(* IEC 61131-3 sources: volt/packages/volt-lsp-iec/test-corpus/lenze-mid/Device/Plc Logic/Application/Library Manager/L_MC4P_RoboticHandling (part 2) *)

(* ---- AXES_GROUP_KIN.pou ---- *)
FUNCTION_BLOCK AXES_GROUP_KIN EXTENDS AXES_GROUP_REF
VAR_INPUT
	AGBC_INT : L_MC4P_AxesGroupBasicControl_internal;
	PICKANDPLACEMEMORY : L_MC4P_PickAndPlaceMemory;
	XENABLEPRECONTROL : BOOL := FALSE;
	FBKINCOORDPROVIDERTMPUSE : L_MC4P_KinCoordProvider;
	FBPG : L_MC1P_PosProfiler;
	FBFBPOOLCOLLECTION : L_UBUP_FBPoolCollection;
	ITFFBPOOL : L_UBUP_IFBPool := fbFBPoolCollection;
	ITFJOBRECEIVER : L_UBUP_IJobReceiver;
END_VAR
VAR_OUTPUT
	PAXIS_X : POINTER TO AXIS_REF_VMA;
	PAXIS_Y : POINTER TO AXIS_REF_VMA;
	PAXIS_Z : POINTER TO AXIS_REF_VMA;
	PAXIS_A : POINTER TO AXIS_REF_VMA;
	PAXIS_B : POINTER TO AXIS_REF_VMA;
	PAXIS_C : POINTER TO AXIS_REF_VMA;
	XPATHDYNAMICSAVAILABLE : BOOL;
	LRPATHVELOCITY : LREAL;
	LRPATHACCELERATION : LREAL;
	LRPATHROTVELOCITY : LREAL;
	LRPATHROTACCELERATION : LREAL;
	LRTCPVELOCITY : LREAL;
	LRTCPACCELERATION : LREAL;
	XAXESGROUPISHOMED : BOOL := FALSE;
	XINPOSITION : BOOL := FALSE;
END_VAR
VAR
	SCFBSTORE : L_MC4P_MovePathStore;
	FBMOVEFBPOOL : L_MC4P_MoveFBPool;
	FBAGBCFBPOOL : L_MC4P_AGBCFBPool;
	WCS2MCS : REFERENCE TO L_UMTP_RobotPos;
	MCS2WCS : REFERENCE TO L_UMTP_RobotPos;
	LRACTTIMEOR : REFERENCE TO LREAL;
	LRSETTIMEOR : REFERENCE TO LREAL;
	LRACTTIMEDOR : REFERENCE TO LREAL;
	FBCOORD : L_MC4P_KinCoordProvider;
	FBCOORDACT : L_MC4P_KinCoordProvider;
	XMCSDISPLACEMENTSUPPORTED : BOOL := TRUE;
	XDUALUSELICENSEREQUIRED : BOOL := FALSE;
	XDUALUSELICENSEAVAILABLE : BOOL := FALSE;
	XUSEJACOBI : BOOL := TRUE;
	LWSOURCEOFMOTION : LWORD := 0;
	LWFTRIGSOURCEOFMOTION : LWORD := 0;
	XWCSFILTERAVAILABLE : BOOL;
	XUNSTEADYWCSPOS : BOOL;
	ALRUNSTEADYPOSWCS : ARRAY [1..3] OF LREAL;
	FBORFILTERLEGACY : L_MC4P_FilterORLegacy;
	FBORFILTERFAST : L_MC4P_FilterORFast;
	FBORFILTERCOMBINED : L_MC4P_FilterORCombine;
	FBVT : L_MC4P_VirtualTime;
	LRACTTIMEOR_LASTCYCLE : LREAL;
	LROVRREQUESTED : LREAL := 1.0;
	LROVFADINGTIME : LREAL := 0.5;
	_DWOBJID : DWORD;
	PSCTRAFOINFO_SP : POINTER TO L_MC4P_TrafoInfo;
	SCTRAFOINFO_SP : L_MC4P_TrafoInfo;
	PSCTRAFOINFO_ACT : POINTER TO L_MC4P_TrafoInfo;
	SCTRAFOINFO_ACT : L_MC4P_TrafoInfo;
	XPRECONTROLENABLED : BOOL := FALSE;
	AXMCSAXISACTIVE : ARRAY [1..6] OF BOOL;
	AXACSAXISACTIVE : ARRAY [1..6] OF BOOL;
	AXACSAXISALREADYINUSE : ARRAY [1..12] OF BOOL;
	KINPARAMS : L_MC4P_KinematikParam;
	XKINPARAMSVALID : BOOL := FALSE;
	XKINPARAMSVALIDOLD : BOOL := FALSE;
	XKINPARAMSCHANGED : BOOL := FALSE;
	XKINCONFIGAVAILABLE : BOOL := TRUE;
	WINITCOUNTER : WORD;
	ITFKINPARAMS : L_MC4P_IKinematicParameter;
	ITFTRAFO : L_MC4P_ITrafoInterface;
	ITFFFWDTORQUE : L_MC4P_itfTorquePreControl;
	ITFEXTTORQUE : L_MC4P_itfExtDynamics;
	ITFVISU : L_MC4P_VisuInterface;
	ALRTORQUETMP : ARRAY [1..6] OF LREAL;
	AMC_STOP : ARRAY [13..18] OF L_MC1P.L_MC1P_Stop_Internal;
	AMC_HALT : ARRAY [13..18] OF L_MC1P.L_MC1P_Halt_Internal;
	FBDUMMY : L_MC1P.L_MC1P_Template;
	ASCPCSTRACKINGPARAM : ARRAY [1..16] OF L_MC4P_PCSTrackParam;
	DATAVALIDTRACKINGOLD : BOOL := FALSE;
	ECOORDSYSTEMLASTTARGET : L_MC4P_CoordSystem := L_MC4P_CoordSystem.MCS;
	XREAKTONMCFBERROR : BOOL;
	APCS : ARRAY [1..16] OF L_MC4P_CoordTrafo;
	ATOOL : ARRAY [0..4] OF L_MC4P_ToolTrafo;
	AITOOLBUFFERED : ARRAY [0..4] OF INT;
	WACTIVETOOL : L_MC4P_ToolSystem;
	WBUSYTOOL : L_MC4P_ToolSystem;
	MCS : L_MC4P_CoordTrafo;
	AEJCSTRAVERSINGRANGE : ARRAY [1..6] OF L_MC1P_TraversingRange := [6(L_MC1P_TraversingRange.Limited)];
	ALRAPPLVELLIMITS : ARRAY [1..18] OF LREAL := [18(0)];
	ALRAPPLACCLIMITS : ARRAY [1..18] OF LREAL := [18(0)];
	ALRAPPLJERKLIMITS : ARRAY [1..18] OF LREAL := [18(0)];
	WLOOKAHEADHORIZON : WORD;
	XENABLEFULLBLENDING : BOOL := TRUE;
	XLIMITTANGENTIALROTATION : BOOL;
	LRMAXVELTRANSLATION : LREAL;
	LRMAXACCTRANSLATION : LREAL;
	LRMAXJERKTRANSLATION : LREAL;
	LRMAXVELROTATION : LREAL;
	LRMAXACCROTATION : LREAL;
	LRMAXJERKROTATION : LREAL;
	LRTIMEINLISTMIN : LREAL := 0.5;
	LRLA_SECURECYCLECOUNT : LREAL := 20;
	XSETVALUESAVAILABLE : BOOL := FALSE;
	XUSEREALDRIVESASVIRTUAL : BOOL := FALSE;
	XUSEREALDRIVESASVIRTUALOLD : BOOL := FALSE;
	XWAITFORREALDRIVESDISABLED : BOOL;
	PREPAREPATH : L_MC4P_PreparePath;
	INTERPOLATEPATH : L_MC4P_InterpolatePath;
	XLIMITPATHTOMAINAXES : BOOL := TRUE;
	XINTERRUPTATNEXTBUFFEREDPOS : BOOL := FALSE;
	XERRORSTOPDONE : BOOL;
	AEAXISTYPE : ARRAY [1..24] OF L_MC4P_AxisType := [24(L_MC4P_AxisType.unconnected)];
	ALRSCALEGENERALIZEDFORCETOTORQUE : ARRAY [1..6] OF LREAL := [6(1)];
	ALRSCALETORQUETOGENERALIZEDFORCE : ARRAY [1..6] OF LREAL := [6(1)];
	USINBROFACSAXES : USINT;
	EROTATIONCONVENTION : L_UMTP_RotationConvention := L_UMTP_RotationConvention.XYZ_rotated;
	AXROTANGLESFIXED : ARRAY [1..3] OF BOOL := [FALSE, FALSE, FALSE];
	WGROUPSTATUS : DWORD := 0;
	XSETINPOSITION : BOOL;
	PCONNECTOR_AXIS_X : POINTER TO IoConfigConnector;
	PCONNECTOR_AXIS_Y : POINTER TO IoConfigConnector;
	PCONNECTOR_AXIS_Z : POINTER TO IoConfigConnector;
	PCONNECTOR_AXIS_A : POINTER TO IoConfigConnector;
	PCONNECTOR_AXIS_B : POINTER TO IoConfigConnector;
	PCONNECTOR_AXIS_C : POINTER TO IoConfigConnector;
	APLINKEDAXIS : ARRAY [1..12] OF POINTER TO AXIS_REF;
	ASLINKEDAXISNAME : ARRAY [1..12] OF STRING;
	XACSAXESCONNECTED : BOOL := FALSE;
	XACSAXESCONNECTEDOLD : BOOL := FALSE;
	XGENERICGROUP : BOOL := FALSE;
	PLRDUMMY : POINTER TO LREAL;
	DIRCREATEMOVEPATHDATA : File.DirCreate;
	DIRCREATEDIAGNOSISDATA : File.DirCreate;
	SDIRDIAGNOSISDATA : STRING;
	EJERKMODE : WORD;
	XIGNOREJERK_CP : BOOL := FALSE;
	XIGNOREJERK_PTP : BOOL := FALSE;
	XIGNOREJERK_AUX : BOOL := FALSE;
	DWUNDOBLENDINGCOUNTER : DWORD;
	LRPATHVELOLD : LREAL := 0;
	LRPATHROTVELOLD : LREAL := 0;
	ROTQUAT : ARRAY [1..4] OF LREAL;
	ROTQUATOLD : ARRAY [1..4] OF LREAL;
	ROTMAT_A : ARRAY [1..3, 1..3] OF LREAL;
	ROTMAT_B : ARRAY [1..3, 1..3] OF LREAL;
	ROTMAT_C : ARRAY [1..3, 1..3] OF LREAL;
	ROTMAT_A_OLD : ARRAY [1..3, 1..3] OF LREAL;
	ROTMAT_B_OLD : ARRAY [1..3, 1..3] OF LREAL;
	ROTMAT_C_OLD : ARRAY [1..3, 1..3] OF LREAL;
	APUNKT : LREAL;
	BPUNKT : LREAL;
	CPUNKT : LREAL;
	FBMCDIAGNOSTIC : L_MC4P_MoveFBDiagnostic;
	FBPATHLISTDIAGNOSTIC : L_MC4P_PathListDiagnostic;
	FBTRACELIST : L_MC4P_TraceList;
	FBOBSERVELIMITS : L_MC4P_ObserveLimits;
	DWRUNTIMECNTR : DWORD;
	SCSUPERPOSDATA : L_MC4P_SuperposHandler;
	SCTRACKINGHANDSHAKE : L_MC4P_TrackingHandshake;
	XORIENTATIONCHANGED : BOOL;
	ACSACC : POINTER TO LREAL;
	ACSPOS : POINTER TO LREAL;
	ACSVEL : POINTER TO LREAL;
	ACTIVELIMITS_1 : DWORD;
	ACTIVELIMITS_2 : DWORD;
	ACTUALINTERPOLATEDMOVEFBINSTANCE : STRING;
	ACTUALINTERPOLATEDSEGMENTID : DINT;
	ACTUALINTERPOLATEDSEGMENTTARGETACS : ARRAY [1..6] OF LREAL;
	ACTUALINTERPOLATEDSEGMENTTARGETAUX : ARRAY [1..6] OF LREAL;
	ACTUALINTERPOLATEDSEGMENTTARGETMCS : ARRAY [1..6] OF LREAL;
	ACTUALINTERPOLATEDSEGMENTTARGETWCS : ARRAY [1..6] OF LREAL;
	ACTUALINTERPOLATEDSEGMENTTYPE : L_MC4P_SegmentType;
	ACTUALSEGMENTSTARTPOSWCS : ARRAY [1..6] OF LREAL;
	CHECKWORKSPACE : BOOL;
	CHECKWORKSPACESTEPS : UDINT;
	CLASSID : DINT;
	CONFIGURATION : ARRAY [1..6] OF INT;
	COORDSYSTEMLASTTARGET : L_MC4P_CoordSystem;
	DIGITALSWITCHHANDLER : L_MC4P_IDigSwitchHandling;
	DIM : UDINT;
	ENABLEMCDIAGNOSTIC : BOOL;
	ENABLEOBSERVELIMITS : BOOL;
	ENABLETRACELISTVISU : BOOL;
	FCSACC : POINTER TO LREAL;
	FCSFRAME : POINTER TO L_UMTP_RobotFrame;
	FCSPOS : POINTER TO LREAL;
	FCSVEL : POINTER TO LREAL;
	HOLDOBSERVEDLIMITS : BOOL;
	IGNOREOVERRIDEWAITTIME : BOOL;
	INTERRUPTATNEXTBUFFEREDPOS : BOOL;
	INTERRUPTEDATNEXTBUFFEREDPOS : BOOL;
	JCSACC : POINTER TO LREAL;
	JCSPOS : POINTER TO LREAL;
	JCSVEL : POINTER TO LREAL;
	LA_SECURECYCLECOUNT : LREAL;
	LOWERSYSTEM : UDINT;
	MAXTANGENTROTACC : LREAL;
	MAXTANGENTROTVEL : LREAL;
	MCSACC : POINTER TO LREAL;
	MCSFRAME : POINTER TO L_UMTP_RobotFrame;
	MCSPOS : POINTER TO LREAL;
	MCSVEL : POINTER TO LREAL;
	OBJECTID : DWORD;
	ORIENTATIONCHANGED : BOOL;
	OVRTYPE : L_MC4P_OVRType;
	PATHACCREDUCTIONFACTOR : LREAL;
	PATHLENGTH : LREAL;
	PATHLISTDIAGBUSY : BOOL;
	PATHLISTDIAGDONE : BOOL;
	PATHLISTDIAGENABLE : BOOL;
	PATHLISTDIAGERRORDETECTED : BOOL;
	PATHLISTDIAGNUMOFLISTELEMENTS : INT;
	PATHLISTDIAGREADERRORFILEEXECUTE : BOOL;
	PATHLISTDIAGWRITEFILEBUSY : BOOL;
	PATHLISTDIAGWRITEFILEDONE : BOOL;
	PATHLISTDIAGWRITEFILEERROR : BOOL;
	PATHLISTDIAGWRITEFILEEXECUTE : BOOL;
	REMAININGPATHLENGTH : LREAL;
	REMAININGSEGMENTLENGTH : LREAL;
	RESETOBSERVEDLIMITS : BOOL;
	SEGMENTLENGTH : LREAL;
	STARTWRITINGDIAGNOSTICFILE : BOOL;
	TANGENTIALTRACKINGENABLEPATHREDUCTION : BOOL;
	TIMEINPATHLISTMIN : LREAL;
	TIMEMEASUREMENT : BOOL;
	UPPERSYSTEM : UDINT;
	USEJACOBI : BOOL;
	WCSACC : POINTER TO LREAL;
	WCSFRAME : POINTER TO L_UMTP_RobotFrame;
	WCSPOS : POINTER TO LREAL;
	WCSVEL : POINTER TO LREAL;
	WRITEDIAGNOSTICFILEDONE : BOOL;
END_VAR
END_FUNCTION_BLOCK

METHOD GENERATEHOMINGSTATEAXIS
VAR_INPUT
	XAXESGROUPISHOMEDOLD : BOOL;
END_VAR
END_METHOD

METHOD GETTRACKINGPCS : POINTER TO L_MC4P_PCSTrackParam
VAR_INPUT
	COORDSYSTEM : L_MC4P_CoordSystem;
END_VAR
END_METHOD

METHOD HASAUXAXIS : BOOL
END_METHOD

METHOD HASONLYCROTATION : BOOL
END_METHOD

METHOD HASROTATIONAXIS : BOOL
END_METHOD

METHOD SETCOMMANDEDPOSITION
VAR_IN_OUT
	ALRCOMMANDEDPOSWCS : ARRAY [1..6] OF LREAL;
	ALRCOMMANDEDPOSACS : ARRAY [1..6] OF LREAL;
	ALRCOMMANDEDPOSAUX : ARRAY [1..6] OF LREAL;
END_VAR
END_METHOD

METHOD SETEXTTORQUEITF : L_IE1P_Error
VAR_INPUT
	ITFEXTTORQUE : L_MC4P_itfExtDynamics;
END_VAR
END_METHOD

METHOD SETINPOSPREPARE
END_METHOD

METHOD SETINPOSITION
VAR_INPUT
	XDONE : BOOL;
END_VAR
END_METHOD

METHOD SETKINREF
VAR_INPUT
	KINTRANSFORM : MC_KIN_REF;
END_VAR
END_METHOD

METHOD SETKINTRANSFORM
VAR_INPUT
	TRAFO : L_MC4P_ITrafoInterface;
END_VAR
END_METHOD

METHOD SETPATHINFO
END_METHOD

METHOD SETSTATUSWORD
END_METHOD

METHOD SETTORQUECTRLFB
VAR_INPUT
	FB : L_MC4P_itfTorquePreControl;
END_VAR
END_METHOD

METHOD SETVISUFB
VAR_INPUT
	VISU : L_MC4P_VisuInterface;
END_VAR
END_METHOD

METHOD UPDATESCALEGENERALIZEDFORCETOTORQUE
END_METHOD

METHOD CHECKAXESTRAVERSINGRANGE : L_IE1P_Error
END_METHOD

METHOD CHECKDUALUSE : BOOL
END_METHOD

METHOD CONFIGUREAXESGROUP
END_METHOD

METHOD GETCONFIGURATIONMAINAXIS
VAR_INPUT
	PFATHER : POINTER TO IoConfigConnector;
	NCOUNT : DINT;
END_VAR
END_METHOD

METHOD ADDACSAXESTOGROUP
VAR_INPUT
	WINDEX : WORD;
END_VAR
END_METHOD

METHOD ADDALLMCSAXISTOGROUP
END_METHOD

METHOD CHECKACSCONFIG : BOOL
END_METHOD

METHOD CONFIGUREAXES : L_IE1P_Error
END_METHOD

METHOD GETAXISMCS : BOOL
VAR_INPUT
	PAXISCONNECTOR : POINTER TO IoConfigConnector;
	XCONNECTED : BOOL;
END_VAR
VAR_OUTPUT
	PAXIS : POINTER TO _AXIS_REF_VMA;
END_VAR
END_METHOD

METHOD REGISTERACSAXISINGROUP
VAR_INPUT
	WINDEX : WORD;
END_VAR
END_METHOD

METHOD SETLINKEDAXIS
VAR_INPUT
	WINDEX : WORD;
END_VAR
END_METHOD

METHOD UPDATEVIRTUALMODEACS
VAR_INPUT
	PAXIS : POINTER TO AXIS_REF;
	XVIRTUALMODE : BOOL;
END_VAR
END_METHOD

METHOD MEMORISEIPOVALUES
VAR_INPUT
	ECOORDSYSTEM : L_MC4P_CoordSystem;
END_VAR
END_METHOD

METHOD BACKWARDTRANSFORMATIONTOAXES : L_IE1P_Error
END_METHOD

METHOD BACKWARDTRANSFORMATIONTOAXES_LEGACY : L_IE1P_Error
VAR_OUTPUT
	SCERROR : L_MC4P_ErrorStruct;
END_VAR
VAR_IN_OUT
	FBCOORD : L_MC4P_KinCoordProvider;
END_VAR
END_METHOD

METHOD BACKWARDTRANSFORMATIONTOAXES_USEJACOBI : L_IE1P_Error
VAR_OUTPUT
	SCERROR : L_MC4P_ErrorStruct;
END_VAR
VAR_IN_OUT
	FBCOORD : L_MC4P_KinCoordProvider;
END_VAR
END_METHOD

METHOD CHECKPLAUSIBILITYOFSETVALUES : L_IE1P.L_IE1P_Error
END_METHOD

METHOD CLEARTRACKINGPCSFLAGS
END_METHOD

METHOD CLEARTRACKINGSUPERPOSDATA
END_METHOD

METHOD FORWARDTRANSFORMATIONTOAXES : L_IE1P_Error
VAR_INPUT
	XUSESETVALUES : BOOL;
END_VAR
END_METHOD

METHOD FORWARDTRANSFORMATIONTOAXES_LEGACY : L_IE1P_Error
VAR_INPUT
	XUSESETVALUES : BOOL;
END_VAR
VAR_OUTPUT
	SCERROR : L_MC4P_ErrorStruct;
END_VAR
VAR_IN_OUT
	FBCOORD : L_MC4P_KinCoordProvider;
END_VAR
END_METHOD

METHOD FORWARDTRANSFORMATIONTOAXES_USEJACOBI : L_IE1P_Error
VAR_INPUT
	XUSESETVALUES : BOOL;
END_VAR
VAR_OUTPUT
	SCERROR : L_MC4P_ErrorStruct;
END_VAR
VAR_IN_OUT
	FBCOORD : L_MC4P_KinCoordProvider;
END_VAR
END_METHOD

METHOD GETCOORDTRAFO : POINTER TO L_MC4P_CoordTrafo
VAR_INPUT
	COORDSYSTEM : L_MC4P_CoordSystem;
END_VAR
END_METHOD

METHOD HANDLEUNSTEADYWCSPOS
END_METHOD

METHOD SETUNSTEADYWCSPOS
VAR_INPUT
	ALRUNSTEADYDISTANCE : ARRAY [1..3] OF LREAL;
END_VAR
END_METHOD

METHOD SUPERPOSETRACKINGVALUES
END_METHOD

METHOD TRACKINGSETSETVALUESAVAILABLE
END_METHOD

METHOD GETMAXACCELERATION : LREAL
VAR_INPUT
	IDX : UINT;
	EMAXVALUESOURCE : L_MC4P_MaxValueSource;
END_VAR
END_METHOD

METHOD GETMAXDECELERATION : LREAL
VAR_INPUT
	IDX : UINT;
	EMAXVALUESOURCE : L_MC4P_MaxValueSource;
END_VAR
END_METHOD

METHOD GETMAXJERK : LREAL
VAR_INPUT
	IDX : UINT;
	EMAXVALUESOURCE : L_MC4P_MaxValueSource;
END_VAR
END_METHOD

METHOD GETMAXVELOCITY : LREAL
VAR_INPUT
	IDX : UINT;
	EMAXVALUESOURCE : L_MC4P_MaxValueSource;
END_VAR
END_METHOD

METHOD EQUALS : BOOL
VAR_INPUT
	ITFPROVIDER : L_MC4P_IKinCoordProvider;
	UDISYSTEM : UDINT;
	XPOS : BOOL;
	XVEL : BOOL;
	XACC : BOOL;
END_VAR
END_METHOD

METHOD REQUESTINTERFACE : BOOL
VAR_INPUT
	ID : DINT;
	PITFUNKNOWN : POINTER TO L_UBUP_IUnknown;
END_VAR
END_METHOD

METHOD SETINSTANCESTRINGMOVEPATHSTORE
VAR_INPUT
	SINSTANCESTR : STRING;
END_VAR
END_METHOD

METHOD APPLYOVERRIDE
VAR_IN_OUT
	LRVEL : LREAL;
	LRACC : LREAL;
END_VAR
END_METHOD

METHOD SETTIMEOVERRIDE
VAR_INPUT
	LROVERRIDE : LREAL;
	LRFADINGTIME : LREAL;
END_VAR
END_METHOD

METHOD CALCSCALEFUNCTIONS
VAR_INPUT
	OFFSET : DWORD;
	INDEX : WORD;
END_VAR
END_METHOD

METHOD CHECKPARAMETER : BOOL
END_METHOD

METHOD ISACTIVEMOTIONCOMMAND : BOOL
VAR_INPUT
	ESRCOFCMD : L_MC4P_SourceOfMotionCommand;
END_VAR
END_METHOD

METHOD RELEASEMOTIONCOMMAND : BOOL
VAR_INPUT
	ESRCOFCMD : L_MC4P_SourceOfMotionCommand;
END_VAR
END_METHOD

METHOD REQUESTMOTIONCOMMAND : L_IE1P_Error
VAR_INPUT
	ESRCOFCMD : L_MC4P_SourceOfMotionCommand;
END_VAR
END_METHOD

METHOD RESETSOURCEOFMOTION
END_METHOD

METHOD SETVALUESCALCULATED
END_METHOD

METHOD UPDATESOURCEOFMOTIONCOMMAND : BOOL
END_METHOD

METHOD CALLSTOPPINTERPOLATOR
VAR_INPUT
	LRINPUTDECELERATION : LREAL;
	LRINPUTJERK : LREAL;
END_VAR
VAR_OUTPUT
	XERROR : BOOL;
	EERRORID : L_IE1P_Error;
	DWINTERNALID : DWORD;
	XDONE : BOOL;
END_VAR
END_METHOD

METHOD ERRORSTOP
END_METHOD

METHOD HALTAUX : BOOL
VAR_OUTPUT
	XERROR : BOOL;
END_VAR
END_METHOD

METHOD LEAVEERRORSTOP
END_METHOD

METHOD LEAVEERRORSTOPPREPARE : BOOL
VAR_INPUT
	XLEAVEERRORSTOP : BOOL;
END_VAR
END_METHOD

METHOD STOPAUX : BOOL
VAR_OUTPUT
	XERROR : BOOL;
END_VAR
END_METHOD

METHOD GETPATHCOORDINATESYSTEM
VAR_OUTPUT
	ALRTANGENT : ARRAY [1..3] OF LREAL;
	ALRNORMAL : ARRAY [1..3] OF LREAL;
	ALRBINORMAL : ARRAY [1..3] OF LREAL;
END_VAR
END_METHOD

METHOD BUFFERTOOL : BOOL
VAR_INPUT
	ETOOLSYSTEM : L_MC4P_ToolSystem;
END_VAR
END_METHOD

METHOD CALCTOOLDISTANCE : BOOL
VAR_INPUT
	ETOOL1 : L_MC4P_ToolSystem;
	ETOOL2 : L_MC4P_ToolSystem;
	SCFCSFRAME : REFERENCE TO L_UMTP_RobotFrame;
	SCDISTWCS : REFERENCE TO L_UMTP_RobotPos;
	SCDISTFCS : REFERENCE TO L_UMTP_RobotPos;
END_VAR
END_METHOD

METHOD CLEARTOOLBUFFER : BOOL
END_METHOD

METHOD GETTOOL : POINTER TO L_MC4P_ToolTrafo
VAR_INPUT
	TOOLSYSTEM : L_MC4P_ToolSystem;
END_VAR
END_METHOD

METHOD SETACTIVETOOL : BOOL
VAR_INPUT
	ETOOLSYSTEM : L_MC4P_ToolSystem;
END_VAR
VAR_OUTPUT
	XTOOLCHANGED : BOOL;
END_VAR
END_METHOD

METHOD TOOLPARAMAPPLICABLE : L_IE1P_Error
VAR_INPUT
	ETOOLSYSTEM : L_MC4P_ToolSystem;
	SCTOOLPARAMETER : L_MC4P_TOOL_REF;
END_VAR
END_METHOD

METHOD TOOLROTATIONISIDENTITY : BOOL
VAR_INPUT
	ETOOLSYSTEM : L_MC4P_ToolSystem;
END_VAR
END_METHOD

METHOD AFTERREADINPUTS : INT
END_METHOD

METHOD AFTERWRITEOUTPUTS
END_METHOD

METHOD BEFOREREADINPUTS : INT
END_METHOD

METHOD BEFOREWRITEOUTPUTS
END_METHOD

METHOD CALL_WCSBWO
END_METHOD

METHOD FB_EXIT : BOOL
VAR_INPUT
	BINCOPYCODE : BOOL;
END_VAR
END_METHOD

METHOD INITFORSIMULATIONMODE : BOOL
VAR_INPUT
	WMODULETYPE : UINT;
	DWINSTANCE : UDINT;
	PCONNECTOR : POINTER TO IoConfigConnector;
END_VAR
END_METHOD

METHOD INITIALIZE : UDINT
VAR_INPUT
	WMODULETYPE : UINT;
	DWINSTANCE : UDINT;
	PCONNECTOR : POINTER TO IoConfigConnector;
END_VAR
END_METHOD

METHOD IODRVREADPARAMETER : UDINT
VAR_INPUT
	PCONNECTOR : POINTER TO IoConfigConnector;
	PPARAMETER : POINTER TO IoConfigParameter;
	PDATA : POINTER TO BYTE;
	DWBITSIZE : DWORD;
	DWBITOFFSET : DWORD;
END_VAR
END_METHOD

METHOD IODRVUPDATECONFIGURATION : UDINT
VAR_INPUT
	PCONNECTORLIST : POINTER TO IoConfigConnector;
	NCOUNT : DINT;
END_VAR
END_METHOD

METHOD IODRVWRITEPARAMETER : UDINT
VAR_INPUT
	PCONNECTOR : POINTER TO IoConfigConnector;
	PPARAMETER : POINTER TO IoConfigParameter;
	PDATA : POINTER TO BYTE;
	DWBITSIZE : DWORD;
	DWBITOFFSET : DWORD;
END_VAR
END_METHOD

METHOD FB_INIT : BOOL
VAR_INPUT
	BINITRETAINS : BOOL;
	BINCOPYCODE : BOOL;
END_VAR
END_METHOD

(* ---- AXES_GROUP_REF.pou ---- *)
FUNCTION_BLOCK AXES_GROUP_REF EXTENDS AXES_GROUP_BASE
VAR_INPUT
	EAXESGROUPSTATE : L_MC4P_AxesGroup_State := L_MC4P_AxesGroup_State.GroupDisabled;
	XGROUPENABLE : BOOL;
	ASCERRORINFO : REFERENCE TO ARRAY [0..7] OF L_IE1P_ErrorInformation;
	ASCWARNINGINFO : REFERENCE TO ARRAY [0..7] OF L_IE1P_ErrorInformation;
	FBFUNIDMANAGER : L_MC4P_FunIDManager;
END_VAR
VAR_OUTPUT
	XERROR : BOOL := FALSE;
	XWARNING : BOOL := FALSE;
	EACTIVEERRORID : L_IE1P_Error;
	XGROUPENABLED : BOOL;
	AXESGROUPNAME : STRING;
END_VAR
VAR
	SCPARAMS : L_MC4P_AxesGroupMember;
	XWRITEGROUPPARAMETERDISABLED : BOOL;
	XISAXES_GROUP_KIN : BOOL := FALSE;
	EKINEMATIC : L_MC4P_KinematicType;
	APAXIS : ARRAY [1..18] OF POINTER TO AXIS_REF;
	ERRORMANAGER : L_IE1P_ErrorManager;
	ERRORRESETOCCUREDTIMEWITHOUTLEM : SYSTIME;
	DWGROUPERRORITFID : DWORD;
	ADWAXISERRORITFID : ARRAY [1..18] OF DWORD;
	PSERRORINST : POINTER TO STRING;
	SERRORINST : STRING;
	XENABLELOGENTRY : BOOL := TRUE;
	EAXESGROUPSTATEOLD : L_MC4P_AxesGroup_State := L_MC4P_AxesGroup_State.GroupDisabled;
	SINSTANCESTR : STRING;
	PATHLIST : L_MC4P_PathDataList;
	LRTASKCYCLE : LREAL := 0.001;
	DWTASKYCLE_US : DWORD := 1000;
	LRINVTASKCYCLE : LREAL := 1000;
	DWCALLCYCLE : DWORD;
	DWCALLCYCLE_US : DWORD;
	XCONNECTORDISABLED : BOOL;
	WINITSTATE : WORD := 0;
	ITFPARA : L_MC1P_IPara;
	AWPOWID : ARRAY [1..6] OF WORD := [6(0)];
	DWPARABASEINDEX : DWORD;
	PPARA2 : L_SSYP.L_SSYP_EVTPARAM_CmpLenzeIPCSystemSoftPLCParaChanged;
	HEVENTPARWRITE : Systypes.RTS_IEC_HANDLE;
	HINTERFACEPARWRITE : Systypes.RTS_IEC_HANDLE;
	HEVENTDOWNLOADDONE : Systypes.RTS_IEC_HANDLE;
	HINTERFACEDOWNLOADDONE : Systypes.RTS_IEC_HANDLE;
	HEVENTRESETDONE : Systypes.RTS_IEC_HANDLE;
	HINTERFACERESETDONE : Systypes.RTS_IEC_HANDLE;
	ITFCALLBACK : CmpEventMgr.ICmpEventCallback;
	DWEVENTCOUNTER : DWORD;
	XENABLEGROUPBLOCKEDBYOBJECTTRANSFER : BOOL;
	DWEVTINITCOUNT : DWORD := 0;
	DWPREINITCOUNT : DWORD := 0;
	STARTTIME : TIME;
	SCTIMESTAMP : L_MC1P_TimeStamp;
	XACTIVATETIMEMEASUREMENT : BOOL := FALSE;
	SCPAR : L_MC4P_ParAccess;
	XREFDUMMY : BOOL;
	LRREFDUMMY : LREAL;
	RREFDUMMY : REAL;
	WREFDUMMY : WORD;
	IREFDUMMY : INT;
	DWREFDUMMY : DWORD;
	DIREFDUMMY : DINT;
	LWREFDUMMY : LWORD;
	LIREFDUMMY : LINT;
	SREFDUMMY : STRING;
	USIREFDUMMY : USINT;
	UIREFDUMMY : UINT;
	UDIREFDUMMY : UDINT;
	ULIREFDUMMY : ULINT;
	MODULEHANDLERBASE : L_IMHP_ModuleHandler := STRUCT(CompActiveDefault := FALSE, Layer := L_IMHP_Layer.Kinematics, CompType := L_IMHP_ComponentType.RobotKinematic);
	HEVENTRESETOCCURED : Systypes.RTS_IEC_HANDLE := SysTypes.RTS_INVALID_HANDLE;
	HINTERFACERESETOCCURED : Systypes.RTS_IEC_HANDLE := SysTypes.RTS_INVALID_HANDLE;
	WEVTCOUNT_RESETOCCURED : WORD;
	XINTERNALERRORRESET : BOOL;
	XINTERNALERRORRESETFROMLEM : BOOL;
	FBBASE : L_MC4P_Template_ForAG;
	GROUPRESETINTERNAL : L_MC4P_GroupReset_Internal;
	XPREPARELEAVEERRORSTOP : BOOL;
	SCERRORSTOPCMD : L_MC1P_StopOperation;
	AEPARAMETERINDEX : ARRAY [1..4] OF L_MC4P_ParameterIndex := [L_MC4P_ParameterIndex.OneOfFour, L_MC4P_ParameterIndex.TwoOfFour, L_MC4P_ParameterIndex.ThreeOfFour, L_MC4P_ParameterIndex.FourOfFour];
	C_STRNOERROR : STRING := '-';
	C_STRUNDEFERROR : STRING := 'undefined';
	LICENSECONFIG : STRING;
	MODULEHANDLER : L_IMHP_IModuleHandler;
END_VAR
END_FUNCTION_BLOCK

METHOD ADDAXISTOGROUP
VAR_INPUT
	PAXIS : POINTER TO AXIS_REF;
	WIDENTINGROUP : WORD;
END_VAR
END_METHOD

METHOD CALLERRORRESETFORALLCOMPONENTS : DINT
END_METHOD

METHOD CHECKPARAMETER : BOOL
END_METHOD

METHOD CLEARERROR
VAR_INPUT
	INSTANCEID : DWORD := 0;
END_VAR
END_METHOD

METHOD CLEARERRORID
VAR_INPUT
	INSTANCEID : DWORD := 0;
	WERRORID : WORD;
END_VAR
END_METHOD

METHOD CLEARERRORID2
VAR_INPUT
	INSTANCEID : DWORD := 0;
	WERRORID : WORD;
	DWEXTENDEDERRORINFO : DWORD;
END_VAR
END_METHOD

METHOD CONFIGUREAXESGROUP
END_METHOD

METHOD ENABLEMAINAXIS : L_IE1P_Error
VAR_INPUT
	XENABLE : BOOL;
END_VAR
VAR_OUTPUT
	STATUS : BOOL;
	VALID : BOOL;
	ERROR : BOOL;
	ERRORID : L_IE1P_Error;
END_VAR
END_METHOD

METHOD GETERRORITFID : DWORD
END_METHOD

METHOD GROUPENABLE
END_METHOD

METHOD HANDLEERRORENTRY : DINT
VAR_INPUT
	WERRORID : L_IE1P_Error := L_IE1P_Error.NoError;
	INSTANCEID : DWORD := 0;
	PSINSTANCENAME : POINTER TO BYTE := 0;
	ESEVERITY : L_IE1P_SeverityLevel := 0;
	DWINTERNALID : DWORD := 0;
	XAUTORESET : BOOL := FALSE;
	XNOLOGGINGENTRY : BOOL := FALSE;
	XEXTERNALERROR : BOOL;
END_VAR
END_METHOD

METHOD NOTIFYERROR
VAR_INPUT
	WERRORID : L_IE1P_Error := L_IE1P_Error.NoError;
	INSTANCEID : DWORD := 0;
	PSINSTANCENAME : POINTER TO BYTE := 0;
	XSETERRORSTOP : BOOL := FALSE;
	DWINTERNALID : DWORD := 0;
END_VAR
END_METHOD

METHOD NOTIFYERRORAXIS
VAR_INPUT
	IDX : WORD;
	WERRORID : L_IE1P_Error;
	EERRORREACTION : L_IE1P_SeverityLevel;
END_VAR
END_METHOD

METHOD EVENTCALLBACK : UDINT
VAR_INPUT
	PEVENTPARAM : POINTER TO EventParam;
END_VAR
END_METHOD

METHOD REGISTEREVENT
END_METHOD

METHOD UNREGISTEREVENT
END_METHOD

METHOD ITFCHECKERRORRESETOCCURED : BOOL
VAR_IN_OUT
	RESETTIME : SYSTIME;
END_VAR
END_METHOD

METHOD ITFCLEARERROR : DWORD
VAR_INPUT
	ESEVERITY : L_IE1P_SeverityLevel;
	WERRORID : WORD;
	WCOMPID : WORD;
	DWINSTANCEID : DWORD := 0;
END_VAR
END_METHOD

METHOD ITFCLEARREACTION
VAR_INPUT
	EREACTION : L_IE1P_Reaction;
	DICLEARCOUNT : DINT;
	DWINSTANCEID : DWORD;
END_VAR
END_METHOD

METHOD ITFGETACTUALERRORCODE : DWORD
VAR_OUTPUT
	ESEVERITY : WORD;
END_VAR
END_METHOD

METHOD ITFREGISTERERRORINSTANCE : DWORD
END_METHOD

METHOD ITFRESETACTIVE : BOOL
END_METHOD

METHOD ITFRESETERROR : DWORD
VAR_INPUT
	ERRORHANDLE : SysTypes.RTS_IEC_HANDLE := 0;
END_VAR
END_METHOD

METHOD ITFRESETERRORREACTION
VAR_INPUT
	DWINSTANCEID : DWORD := 0;
END_VAR
END_METHOD

METHOD ITFSETERROR : DWORD
VAR_INPUT
	ESEVERITY : L_IE1P_SeverityLevel;
	WERRORID : WORD;
	WCOMPID : WORD;
	DWINSTANCEID : DWORD := 0;
	EREACTION : L_IE1P_Reaction;
END_VAR
END_METHOD

METHOD CALCSCALEFUNCTIONS
VAR_INPUT
	OFFSET : DWORD;
	INDEX : WORD;
END_VAR
END_METHOD

METHOD HLP_GETPARAMETER : BOOL
END_METHOD

METHOD HLP_GETPARAMETERPROPERTIES : BOOL
VAR_INPUT
	DIPARAMETER : DINT;
END_VAR
VAR_OUTPUT
	PPARAMADDR : POINTER TO BYTE := 0;
	EORDINALTYPE : L_MC1P_OrdinalType := L_MC1P_OrdinalType.otNONE;
	XREADWRITE : BOOL := FALSE;
	LRUNITFACTOR : LREAL := 1.0;
	LRDEFAULTVALUE : LREAL := 0.0;
	WVALUERANGES : WORD := 0;
	PVALUERANGES : POINTER TO L_MC1P_MinMaxValue := 0;
END_VAR
END_METHOD

METHOD HLP_INITPARREF
END_METHOD

METHOD HLP_READBOOLPARAMETER : BOOL
VAR_INPUT
	PARAMETER : DINT;
	PXVALUE : POINTER TO BOOL;
END_VAR
END_METHOD

METHOD HLP_READPARAMETER : BOOL
VAR_INPUT
	PARAMETER : DINT;
	PLRVALUE : POINTER TO LREAL;
END_VAR
END_METHOD

METHOD HLP_WRITEBOOLPARAMETER : BOOL
VAR_INPUT
	PARAMETER : DINT;
	PXVALUE : POINTER TO BOOL;
END_VAR
VAR_OUTPUT
	WERRORID : WORD;
END_VAR
END_METHOD

METHOD HLP_WRITEPARAMETER : BOOL
VAR_INPUT
	PARAMETER : DINT;
	PLRVALUE : POINTER TO LREAL;
END_VAR
VAR_OUTPUT
	WERRORID : WORD;
END_VAR
END_METHOD

METHOD AFTERREADINPUTS : INT
END_METHOD

METHOD AFTERWRITEOUTPUTS
END_METHOD

METHOD BEFOREREADINPUTS : INT
END_METHOD

METHOD BEFOREWRITEOUTPUTS
END_METHOD

METHOD FB_EXIT : BOOL
VAR_INPUT
	BINCOPYCODE : BOOL;
END_VAR
END_METHOD

METHOD IODRVREADPARAMETER : UDINT
VAR_INPUT
	PCONNECTOR : POINTER TO IoConfigConnector;
	PPARAMETER : POINTER TO IoConfigParameter;
	PDATA : POINTER TO BYTE;
	DWBITSIZE : DWORD;
	DWBITOFFSET : DWORD;
END_VAR
END_METHOD

METHOD IODRVUPDATEMAPPING : UDINT
VAR_INPUT
	PTASKMAPLIST : POINTER TO IoConfigTaskMap;
	NCOUNT : DINT;
END_VAR
END_METHOD

METHOD IODRVWRITEPARAMETER : UDINT
VAR_INPUT
	PCONNECTOR : POINTER TO IoConfigConnector;
	PPARAMETER : POINTER TO IoConfigParameter;
	PDATA : POINTER TO BYTE;
	DWBITSIZE : DWORD;
	DWBITOFFSET : DWORD;
END_VAR
END_METHOD

METHOD QUERYINTERFACE : POINTER TO POINTER TO BYTE
VAR_INPUT
	IID : DWORD;
	PRESULT : POINTER TO UDINT;
END_VAR
END_METHOD

METHOD FB_INIT : BOOL
VAR_INPUT
	BINITRETAINS : BOOL;
	BINCOPYCODE : BOOL;
END_VAR
END_METHOD

(* ---- GLOBALTEXTLIST.pou ---- *)
FUNCTION_BLOCK GLOBALTEXTLIST
VAR
	M_TEXTLISTFILE : STRING(255);
	_STNAMESPACE : STRING;
END_VAR
END_FUNCTION_BLOCK

(* ---- L_MC4P_AGBCFBPOOL.pou ---- *)
FUNCTION_BLOCK L_MC4P_AGBCFBPOOL EXTENDS L_UBUP_FBPool
VAR
	_SCAGBCRESOURCE : REFERENCE TO L_MC4P_AxesGroupBasicControl_internal;
	_XMEMOWNER1 : BOOL;
	_AABCV2 : ARRAY [1..18] OF L_MC1P_AxisBasicControlV2;
	_ABCV2CONTROLNODES : L_UBUP_DoubleLinkedListNodes;
	_ABCV2CONTROL : L_UBUP_DoubleLinkedListControl;
	_GROUPMANUALMODECONTROLNODES : L_UBUP_DoubleLinkedListNodes;
	_GROUPMANUALMODECONTROL : L_UBUP_DoubleLinkedListControl;
	_GROUPHOMECONTROLNODES : L_UBUP_DoubleLinkedListNodes;
	_GROUPHOMECONTROL : L_UBUP_DoubleLinkedListControl;
	_GROUPSTOPCONTROLNODES : L_UBUP_DoubleLinkedListNodes;
	_GROUPSTOPCONTROL : L_UBUP_DoubleLinkedListControl;
	_GROUPREADSTATUSCONTROLNODES : L_UBUP_DoubleLinkedListNodes;
	_GROUPREADSTATUSCONTROL : L_UBUP_DoubleLinkedListControl;
	_GROUPSETOVERRIDECONTROLNODES : L_UBUP_DoubleLinkedListNodes;
	_GROUPSETOVERRIDECONTROL : L_UBUP_DoubleLinkedListControl;
	_GROUPSETPOSITIONCONTROLNODES : L_UBUP_DoubleLinkedListNodes;
	_GROUPSETPOSITIONCONTROL : L_UBUP_DoubleLinkedListControl;
	USEGLOBAL : BOOL;
END_VAR
END_FUNCTION_BLOCK

METHOD FB_INIT : BOOL
VAR_INPUT
	BINITRETAINS : BOOL;
	BINCOPYCODE : BOOL;
	SCAGBCRESOURCE : REFERENCE TO L_MC4P_AxesGroupBasicControl_internal;
END_VAR
END_METHOD

METHOD FREERESOURCE
END_METHOD

METHOD GETFB : L_UBUP_IPoolInstance
VAR_INPUT
	ECLASSID : DINT;
	DWARRIDX : DWORD;
END_VAR
END_METHOD

METHOD GETFBCONTROL : L_UBUP_IListControl
VAR_INPUT
	ECLASSID : DINT;
END_VAR
END_METHOD

METHOD OCCUPYRESOURCE : BOOL
VAR_INPUT
	ECLASSID : DINT;
END_VAR
END_METHOD

METHOD SETCAPACITYALL
END_METHOD

(* ---- L_MC4P_AVGVALUEFILTER1D.pou ---- *)
FUNCTION_BLOCK L_MC4P_AVGVALUEFILTER1D EXTENDS L_UBUP_MemoryProvider
VAR_INPUT
	XENABLE : BOOL;
	UIFILTERTIME : UINT;
	LRVALUEIN : LREAL;
	ETRAVERSINGRANGE : L_MC1P_TraversingRange := L_MC1P_TraversingRange.Limited;
	LRCYCLELENGTH : LREAL;
END_VAR
VAR_OUTPUT
	XBUSY : BOOL;
	XACTIVE : BOOL;
	XERROR : BOOL;
	EERRORID : L_IE1P.L_IE1P_Error;
	DWINTERNALID : DWORD;
	LRVALUEOUT : LREAL;
END_VAR
VAR
	LRTASKCYCLE : LREAL := -1;
	XENABLE_R : R_Trig;
	AMEM : ARRAY [1..cuiFilterSizeMax] OF LREAL;
	FB_AVG : L_USPP_AverageFilterRecursive;
	CUIFILTERSIZEMAX : UINT := 101;
	PTR : POINTER TO BYTE;
	SIZE : UDINT;
END_VAR
END_FUNCTION_BLOCK

(* ---- L_MC4P_AXESGROUPBASICCONTROL.pou ---- *)
FUNCTION_BLOCK L_MC4P_AXESGROUPBASICCONTROL EXTENDS L_MC4P_Template_AG_KIN_Licence
VAR_INPUT
	XENABLEINTERNALCONTROL : BOOL;
	XRESETAXESGROUP : BOOL;
	XREGULATORONALL : BOOL;
	XENABLEAXESGROUP : BOOL;
	LROVERRIDE : LREAL := 1;
	XSTOPALL : BOOL;
	SCPAR : L_MC4P_AGBC_Parameter;
	ECOORDSYSTEM : L_MC4P_CoordSystem := L_MC4P_CoordSystem.WCS;
	XGROUPSTOPEXECUTE : BOOL;
	XMOVEDIRABSEXECUTE : BOOL;
	XMOVEDIRRELEXECUTE : BOOL;
	XMOVELINABSEXECUTE : BOOL;
	XMOVELINRELEXECUTE : BOOL;
	ALRSETPOSDIST : ARRAY [1..12] OF LREAL;
	XGROUPSETPOSEXECUTE : BOOL;
	XGROUPHOMEEXECUTE : BOOL;
	AXHOMEABSSWITCH : ARRAY [1..12] OF BOOL;
	ASCHOMEEXTTP : ARRAY [1..12] OF MC_TRIGGER_REF;
	AXJOGPOS : ARRAY [1..12] OF BOOL;
	AXJOGNEG : ARRAY [1..12] OF BOOL;
	AXMOVEABS : ARRAY [1..12] OF BOOL;
	AXMOVEREL : ARRAY [1..12] OF BOOL;
	ASCCTRLABC : ARRAY [1..18] OF L_MC1P_CtrlABC;
END_VAR
VAR_OUTPUT
	XINTERNALCONTROLACTIVE : BOOL;
	XERROR : BOOL;
	EERRORID : L_IE1P_Error;
	XFUNBUSY : BOOL;
	XFUNDONE : BOOL;
	XFUNCOMMANDABORTED : BOOL;
	EFUNSTATEACT : L_MC4P_AGBC_State := L_MC4P_AGBC_State.Standby;
	XAXESGROUPHOMED : BOOL;
	XHWLIMITSWITCHANY : BOOL;
	XSWLIMITENABLEDALL : BOOL;
	XSWLIMITSWITCHANY : BOOL;
	EKINEMATICTYPE : L_MC4P_KinematicType;
	EAXESGROUPSTATE : L_MC4P_AxesGroup_State;
	XAXESGROUPENABLED : BOOL;
	XREALAXESREADYALL : BOOL;
	XREALAXESENABLEDALL : BOOL;
	XINPOSITION : BOOL;
	XAXESGROUPWARNING : BOOL;
	XAXESGROUPERROR : BOOL;
	EAXESGROUPERRORID : L_IE1P_Error;
	ALRACTPOS : ARRAY [1..12] OF LREAL;
	ALRACTVEL : ARRAY [1..12] OF LREAL;
	ALRSETPOSOUT : ARRAY [1..12] OF LREAL;
	ALRSETVELOUT : ARRAY [1..12] OF LREAL;
	ALRACTFOLLOWINGERROR : ARRAY [1..12] OF LREAL;
	LRSETPATHVELOUT : LREAL;
	LRSETPATHACCOUT : LREAL;
	LRSETTCPACCOUT : LREAL := 0;
	LRSETROTVELOUT : LREAL := 0;
	LRSETROTACCOUT : LREAL := 0;
	ASCSTATUSABC : ARRAY [1..18] OF L_MC1P_StatusABC;
END_VAR
VAR
	XCALLED : BOOL := FALSE;
	XJOGUSEAXESGROUPPAR : BOOL := FALSE;
	JOGUSEAXESGROUPPAR : BOOL;
END_VAR
END_FUNCTION_BLOCK

(* ---- L_MC4P_AXESGROUPBASICCONTROL_INTERNAL.pou ---- *)
FUNCTION_BLOCK L_MC4P_AXESGROUPBASICCONTROL_INTERNAL
VAR_INPUT
	AXHOMEABSSWITCH : ARRAY [1..12] OF BOOL;
	XISV2 : BOOL := FALSE;
END_VAR
VAR_OUTPUT
	XINTERNALCONTROLACTIVE : BOOL;
	XERROR : BOOL;
	EERRORID : L_IE1P_Error;
	XFUNBUSY : BOOL;
	XFUNDONE : BOOL;
	XFUNCOMMANDABORTED : BOOL;
	EFUNSTATEACT : L_MC4P_AGBC_State := L_MC4P_AGBC_State.Standby;
	XAXESGROUPHOMED : BOOL;
	XHWLIMITSWITCHANY : BOOL;
	XSWLIMITENABLEDALL : BOOL;
	XSWLIMITSWITCHANY : BOOL;
	EKINEMATICTYPE : L_MC4P_KinematicType;
	EAXESGROUPSTATE : L_MC4P_AxesGroup_State;
	XAXESGROUPENABLED : BOOL;
	XREALAXESREADYALL : BOOL;
	XREALAXESENABLEDALL : BOOL;
	XAXESGROUPWARNING : BOOL;
	XAXESGROUPERROR : BOOL;
	XINPOSITION : BOOL;
	EAXESGROUPERRORID : L_IE1P_Error;
	ALRACTPOS : ARRAY [1..12] OF LREAL;
	ALRACTVEL : ARRAY [1..12] OF LREAL;
	ALRSETPOSOUT : ARRAY [1..12] OF LREAL;
	ALRSETVELOUT : ARRAY [1..12] OF LREAL;
	ALRACTFOLLOWINGERROR : ARRAY [1..12] OF LREAL;
	LRSETPATHVELOUT : LREAL;
	LRSETPATHACCOUT : LREAL;
	LRSETTCPACCOUT : LREAL := 0;
	LRSETROTVELOUT : LREAL := 0;
	LRSETROTACCOUT : LREAL := 0;
END_VAR
VAR
	FB_SEMAMOVEFBS : L_MC1P_CriticalSection;
	XRESOURCEOWNER : BOOL;
	MC_GROUPRESET1 : MC_GroupReset;
	MC_GROUPENABLE1 : MC_GroupEnable;
	MC_GROUPDISABLE1 : MC_GroupDisable;
	MC_GROUPREADACTUALPOSITION1 : L_MC4P_GroupReadActualPosition_Internal;
	MC_GROUPREADACTUALVELOCITY1 : L_MC4P_GroupReadActualVelocity_Internal;
	MC_GROUPREADERROR1 : MC_GroupReadError;
	MC_GROUPREADSTATUS1 : L_MC4P_GroupReadStatus_Internal;
	MC_GROUPSTOP1 : L_MC4P_GroupStop_Internal;
	MC_GROUPHOME1 : L_MC4P_GroupHome_Internal;
	MC_GROUPSETPOSITION1 : L_MC4P_GroupSetPosition_Internal;
	L_MC4P_GROUPMANUALMODE1 : L_MC4P_GroupManualMode_Internal;
	MC_MOVEDIRECTABSOLUTE1 : L_MC4P_MoveDirectAbsolute_Internal;
	MC_MOVEDIRECTRELATIVE1 : L_MC4P_MoveDirectRelative_Internal;
	MC_MOVELINEARABSOLUTE1 : L_MC4P_MoveLinearAbsolute_Internal;
	MC_MOVELINEARRELATIVE1 : L_MC4P_MoveLinearRelative_Internal;
	L_MC4P_GROUPSETOVERRIDE1 : L_MC4P_GroupSetOverride_Internal;
	AABC : ARRAY [1..18] OF L_MC1P_AxisBasicControl;
	SCPAR_INT : L_MC4P_AGBC_Parameter;
	IDX : WORD;
	WSTOPMODE : WORD;
	ALRSETPOSDIST_INT : ARRAY [1..12] OF LREAL;
	XINTERNALCONTROLVISU : BOOL;
	XRESETAXESGROUP_INT : BOOL;
	XREGULATORONALL_INT : BOOL;
	XENABLEAXESGROUP_INT : BOOL;
	XCOORDMOTIONEXECUTE_INT : BOOL := FALSE;
	XGROUPSTOPEXECUTE_INT : BOOL;
	XSTOPALL_INT : BOOL;
	XGROUPSTOPEXECUTE_INTOREXT : BOOL;
	XMOVEDIRABSEXECUTE_INT : BOOL;
	XMOVEDIRRELEXECUTE_INT : BOOL;
	XMOVELINABSEXECUTE_INT : BOOL;
	XMOVELINRELEXECUTE_INT : BOOL;
	XSTOPALL_INTOREXT : BOOL;
	XSTOPALL_INTOREXTOLD : BOOL;
	XGROUPHOMEEXECUTE_INT : BOOL;
	AXUSEEXTPARAMETER : ARRAY [1..12] OF BOOL;
	XGROUPSETPOSEXECUTE_INT : BOOL;
	AXJOGPOS_INT : ARRAY [1..12] OF BOOL;
	AXJOGNEG_INT : ARRAY [1..12] OF BOOL;
	AXMOVEABS_INT : ARRAY [1..12] OF BOOL;
	AXMOVEREL_INT : ARRAY [1..12] OF BOOL;
	LROVERRIDE_INT : LREAL := 1;
	ECOORDSYSTEM_INT : L_MC4P_CoordSystem := L_MC4P_CoordSystem.MCS;
	DIMAINFRAMESELECT : DINT := 0;
	DIGENERALSUBFRAMESELECT : DINT := 0;
	DIDIAGNOSISFRAMESELECT : DINT := 0;
	DICOORDMOTIONFRAMESELECT : DINT := 0;
	DIHOMINGFRAMESELECT : DINT := 0;
	DIMANMODESELECT : DINT := 0;
	IAXISOFFSETDIAGNOSIS_INT : INT := 0;
	IAUXAXISOFFSET_MANMODE : INT := 0;
	ICOORDSYSOFFSET_MANMODE : INT := 0;
	IAXISOFFSETCOORDMOTION_INT : INT := 0;
	IAXISOFFSETHOMING_INT : INT := 0;
	ESELECTAXISHOMING_INT : IDENT_IN_GROUP_REF := IDENT_IN_GROUP_REF.none;
	ESELECTABC_INT : IDENT_IN_GROUP_REF := IDENT_IN_GROUP_REF.none;
	XSHOWMOVELINPARAMETER : BOOL := FALSE;
	XSHOWMOVEDIRPARAMETER : BOOL := FALSE;
	XSHOWMANMODEPARAMETER : BOOL := FALSE;
	ALRENABLEDORUNCONNECTEDCOLOR : ARRAY [1..30] OF LREAL := [30(16#B0B0B0)];
	ASAXISNAMES : ARRAY [1..30] OF STRING := [30('unconnected')];
	AXAXESAVAILABLE : ARRAY [1..30] OF BOOL;
	XMANMODEVISU_EXECUTE : BOOL;
	XINTERNALCONTROLABCALLOWED : BOOL;
	XINIT : BOOL := TRUE;
	XEXIT : BOOL;
	AXJOGPOSOLD : ARRAY [1..12] OF BOOL;
	AXJOGNEGOLD : ARRAY [1..12] OF BOOL;
	AXMOVEABSOLD : ARRAY [1..12] OF BOOL;
	AXMOVERELOLD : ARRAY [1..12] OF BOOL;
	XGROUPHOMEEXECUTEOLD : BOOL;
	XGROUPSETPOSEXECUTEOLD : BOOL;
	XMOVELINABSEXECUTEOLD : BOOL;
	XMOVELINRELEXECUTEOLD : BOOL;
	XMOVEDIRABSEXECUTEOLD : BOOL;
	XMOVEDIRRELEXECUTEOLD : BOOL;
	XGROUPSTOPEXECUTEOLD : BOOL;
	XRESETAXESGROUPOLD : BOOL;
	XENABLEAXESGROUPOLD : BOOL;
	XFUNDONEOLD : BOOL;
	ECOORDSYSTEMOLD : L_MC4P_CoordSystem;
	PAXESGROUP : POINTER TO AXES_GROUP_KIN := 0;
	XDISABLEMOVEFUNCTIONS : BOOL;
	XAGBC_CALLED : BOOL;
	XAGBC_CALLEDERRORPRESENT : BOOL;
	SINSTANCESTR : STRING;
END_VAR
END_FUNCTION_BLOCK

METHOD EXITSTATE
VAR_IN_OUT
	AXESGROUP : AXES_GROUP_KIN;
	FBBASE : L_MC4P_Template_AG_KIN;
	ASCCTRLABC : ARRAY [1..18] OF L_MC1P_CtrlABC;
END_VAR
END_METHOD

METHOD INIT
VAR_IN_OUT
	AXESGROUP : AXES_GROUP_KIN;
	ASCCTRLABC : ARRAY [1..18] OF L_MC1P_CtrlABC;
END_VAR
END_METHOD

METHOD MAIN
VAR_IN_OUT
	AXESGROUP : AXES_GROUP_KIN;
	FBBASE : L_MC4P_Template_AG_KIN;
	XENABLEINTERNALCONTROL : BOOL;
	XRESETAXESGROUP : BOOL;
	XREGULATORONALL : BOOL;
	XENABLEAXESGROUP : BOOL;
	LROVERRIDE : LREAL;
	XSTOPALL : BOOL;
	SCPAR : L_MC4P_AGBC_Parameter;
	ECOORDSYSTEM : L_MC4P_CoordSystem := L_MC4P_CoordSystem.WCS;
	XGROUPSTOPEXECUTE : BOOL;
	XMOVEDIRABSEXECUTE : BOOL;
	XMOVEDIRRELEXECUTE : BOOL;
	XMOVELINABSEXECUTE : BOOL;
	XMOVELINRELEXECUTE : BOOL;
	ALRSETPOSDIST : ARRAY [1..12] OF LREAL;
	XGROUPSETPOSEXECUTE : BOOL;
	XGROUPHOMEEXECUTE : BOOL;
	ASCHOMEEXTTP : ARRAY [1..12] OF MC_TRIGGER_REF;
	AXJOGPOS : ARRAY [1..12] OF BOOL;
	AXJOGNEG : ARRAY [1..12] OF BOOL;
	AXMOVEABS : ARRAY [1..12] OF BOOL;
	AXMOVEREL : ARRAY [1..12] OF BOOL;
	ASCCTRLABC : ARRAY [1..18] OF L_MC1P_CtrlABC;
	ASCSTATUSABC : ARRAY [1..18] OF L_MC1P_StatusABC;
END_VAR
END_METHOD

METHOD RESETCALLFLAG
END_METHOD

METHOD RESETSTOPMODE
END_METHOD

METHOD SETINSTANCESTRING
VAR_INPUT
	SINSTANCESTR_AXESGROUP : STRING;
END_VAR
END_METHOD

METHOD STATEMACHINE
VAR_IN_OUT
	AXESGROUP : AXES_GROUP_KIN;
	ASCCTRLABC : ARRAY [1..18] OF L_MC1P_CtrlABC;
END_VAR
END_METHOD

METHOD UPDATEVISULAYOUT
VAR_IN_OUT
	AXESGROUP : AXES_GROUP_KIN;
END_VAR
END_METHOD

(* ---- L_MC4P_CALCSTOPPROFILES.pou ---- *)
FUNCTION_BLOCK L_MC4P_CALCSTOPPROFILES
VAR
	XFIRSTSEGMENTOFSTOPSEQUENCE : BOOL;
	XCALCSTOPFAILED : BOOL;
END_VAR
END_FUNCTION_BLOCK

METHOD ADDRESTPHASE
VAR_IN_OUT
	SCPROFILEDATA : L_MC1P_ProfileData;
	LRDESIREDTIME : LREAL;
END_VAR
END_METHOD

METHOD CALCSTOPPROFILES
VAR_INPUT
	LRINPUTDECELERATION : LREAL;
	LRINPUTJERK : LREAL;
END_VAR
VAR_OUTPUT
	XBUSY : BOOL;
	XDONE : BOOL;
	XERROR : BOOL;
	EERRORID : L_IE1P_Error;
	DWINTERNALID : DWORD;
END_VAR
VAR_IN_OUT
	AXESGROUP : AXES_GROUP_KIN;
	FBBASE : L_MC4P_Template_AG_KIN;
END_VAR
END_METHOD

METHOD DECELERATECPSEGMENT
VAR_INPUT
	PLISTELEMENT : POINTER TO L_MC4P_ListElement;
	LRINPUTDECELERATION : LREAL;
	LRINPUTJERK : LREAL;
END_VAR
VAR_OUTPUT
	XSTOPPED : BOOL;
	LRMAXTIME : LREAL;
	XERROR : BOOL;
	EERRORID : L_IE1P_Error;
	DWINTERNALID : DWORD;
END_VAR
VAR_IN_OUT
	AXESGROUP : AXES_GROUP_KIN;
	FBBASE : L_MC4P_Template_AG_KIN;
END_VAR
END_METHOD

METHOD DECELERATEPTPSEGMENT
VAR_INPUT
	PLISTELEMENT : POINTER TO L_MC4P_ListElement;
END_VAR
VAR_OUTPUT
	XSTOPPED : BOOL;
	LRMAXTIME : LREAL;
	XERROR : BOOL;
	EERRORID : L_IE1P_Error;
	DWINTERNALID : DWORD;
END_VAR
VAR_IN_OUT
	AXESGROUP : AXES_GROUP_KIN;
	FBBASE : L_MC4P_Template_AG_KIN;
END_VAR
END_METHOD

METHOD DETERMINEDECELERATION
VAR_INPUT
	LRINPUTDECELERATION : LREAL;
	LRINPUTJERK : LREAL;
	LRPOSSTART : LREAL;
	LRVELSTART : LREAL;
	LRACCSTART : LREAL;
END_VAR
VAR_OUTPUT
	XJUSTSTOPPING : BOOL;
	XERROR : BOOL;
	EERRORID : L_IE1P_Error;
	DWINTERNALID : DWORD;
END_VAR
VAR_IN_OUT
	AXESGROUP : AXES_GROUP_KIN;
	FBBASE : L_MC4P_Template_AG_KIN;
	PROFILEDATAIN : L_MC1P_ProfileData;
	PROFILEPARAMETERIN : L_MC1P_ProfileParameter;
	PROFILEDATAOUT : L_MC1P_ProfileData;
	PROFILEPARAMETEROUT : L_MC1P_ProfileParameter;
END_VAR
END_METHOD

METHOD GETLISTELEMENTTIME : LREAL
VAR_INPUT
	PLE : POINTER TO L_MC4P_ListElement;
END_VAR
END_METHOD

METHOD REVERTLISTCALCSTOPPROFILES : BOOL
VAR_IN_OUT
	AXESGROUP : AXES_GROUP_KIN;
END_VAR
END_METHOD

METHOD SPLITSEGMENT
VAR_INPUT
	PLISTELEMENT : POINTER TO L_MC4P_ListElement;
	PLIST : POINTER TO L_MC4P_PathDataList;
END_VAR
VAR_OUTPUT
	XERROR : BOOL;
	EERRORID : L_IE1P_Error;
	DWINTERNALID : DWORD;
END_VAR
VAR_IN_OUT
	AXESGROUP : AXES_GROUP_KIN;
	FBBASE : L_MC4P_Template_AG_KIN;
END_VAR
END_METHOD

METHOD SYNCDECELERATE : BOOL
VAR_INPUT
	ASCPROFILEDATA : ARRAY [1..6] OF L_MC1P_ProfileData;
	ASCPARAM : ARRAY [1..6] OF L_MC1P_ProfileParameter;
END_VAR
VAR_OUTPUT
	ASCPROFILEDATAOUT : ARRAY [1..6] OF L_MC1P_ProfileData;
	ASCPARAMOUT : ARRAY [1..6] OF L_MC1P_ProfileParameter;
	LRMINTIME : LREAL;
	XERROR : BOOL;
END_VAR
VAR_IN_OUT
	AXESGROUP : AXES_GROUP_KIN;
	FBBASE : L_MC4P_Template_AG_KIN;
END_VAR
END_METHOD

METHOD FINISHCALLBACKS
VAR_INPUT
	PLIST : POINTER TO L_MC4P_PathDataList;
	PLISTELEMENT_ORIGINALEND : POINTER TO L_MC4P_ListElement;
	PLISTELEMENTSTOP : POINTER TO L_MC4P_ListElement;
END_VAR
VAR_OUTPUT
	DWINTERNALID : DWORD;
END_VAR
END_METHOD

(* ---- L_MC4P_CALLTRAFO.pou ---- *)
FUNCTION_BLOCK L_MC4P_CALLTRAFO EXTENDS L_MC4P_Template_AG_KIN
VAR_INPUT
	XENABLE : BOOL;
	ECOORDSYSTEMIN : L_MC4P_CoordSystem;
	ECOORDSYSTEMOUT : L_MC4P_CoordSystem;
	AICONFIG : ARRAY [1..6] OF INT;
	ALRPOSIN : ARRAY [1..6] OF LREAL;
	XVEL : BOOL;
	ALRVELIN : ARRAY [1..6] OF LREAL;
	XACC : BOOL;
	ALRACCIN : ARRAY [1..6] OF LREAL;
END_VAR
VAR_OUTPUT
	XBUSY : BOOL;
	XERROR : BOOL;
	EERRORID : L_IE1P_Error;
	XGIMBALLOCK : BOOL;
	ALRPOSOUT : ARRAY [1..6] OF LREAL;
	ALRVELOUT : ARRAY [1..6] OF LREAL;
	ALRACCOUT : ARRAY [1..6] OF LREAL;
END_VAR
VAR
	_FBCOORD : L_MC4P_KinCoordProvider;
	_SCTRAFOINFO : L_MC4P_TrafoInfo;
	_SCERROR : L_MC4P_ErrorStruct;
	_MODEL : L_UBUP_BehaviourModel_LConC_LENZE;
END_VAR
END_FUNCTION_BLOCK

METHOD CYCLICACTION
VAR_INPUT
	ITFTIMINGCONTROLLER : L_UBUP_ITimingController;
END_VAR
VAR_OUTPUT
	XCOMPLETE : BOOL;
	XABORT : BOOL;
	IERRORID : INT;
END_VAR
END_METHOD

METHOD FINALIZEACTION
VAR_INPUT
	XABORTPROPOSED : BOOL;
	IERRORIDPROPOSED : INT;
END_VAR
VAR_OUTPUT
	XCOMPLETE : BOOL;
	XABORT : BOOL;
	IERRORID : INT;
END_VAR
END_METHOD

METHOD RESETACTION
VAR_OUTPUT
	XCOMPLETE : BOOL;
END_VAR
END_METHOD

METHOD STARTACTION
VAR_OUTPUT
	XCOMPLETE : BOOL;
	IERRORID : INT;
END_VAR
END_METHOD

METHOD FB_INIT : BOOL
VAR_INPUT
	BINITRETAINS : BOOL;
	BINCOPYCODE : BOOL;
END_VAR
END_METHOD

METHOD FB_REINIT : BOOL
END_METHOD

METHOD BWD
VAR_INPUT
	ILOWER : INT;
	IUPPER : INT;
END_VAR
END_METHOD

METHOD CONSISTENCYCHECK : BOOL
VAR_IN_OUT
	AXESGROUP : AXES_GROUP_KIN;
END_VAR
END_METHOD

METHOD COORD2FRAME
VAR_INPUT
	ALRPOSIN : ARRAY [1..6] OF LREAL;
	ALRVELIN : ARRAY [1..6] OF LREAL;
	ALRACCIN : ARRAY [1..6] OF LREAL;
END_VAR
VAR_IN_OUT
	SCROBFRAME : L_UMTP_RobotFrame;
END_VAR
END_METHOD

METHOD COORDSYSTEM2INT : INT
VAR_INPUT
	ESYSTEM : L_MC4P_CoordSystem;
END_VAR
VAR_OUTPUT
	EERRORID : L_IE1P_Error;
END_VAR
END_METHOD

METHOD FWD
VAR_INPUT
	ILOWER : INT;
	IUPPER : INT;
END_VAR
END_METHOD

METHOD PCS2PCS
VAR_INPUT
	ILOWER : INT;
	IUPPER : INT;
END_VAR
END_METHOD

METHOD PCS2WCSFRAME
VAR_INPUT
	IPCS : INT;
	ALRPOSIN : ARRAY [1..6] OF LREAL;
	ALRVELIN : ARRAY [1..6] OF LREAL;
	ALRACCIN : ARRAY [1..6] OF LREAL;
END_VAR
VAR_IN_OUT
	SCP1WCSFRAME : L_UMTP_RobotFrame;
END_VAR
END_METHOD

METHOD PREPARECOORDPROVIDER
VAR_INPUT
	ICOORDSYSTEMIN : INT;
	ICOORDSYSTEMOUT : INT;
END_VAR
END_METHOD

METHOD WCS2PCSFRAME
VAR_INPUT
	IPCS : INT;
	ALRPOSIN : ARRAY [1..6] OF LREAL;
	ALRVELIN : ARRAY [1..6] OF LREAL;
	ALRACCIN : ARRAY [1..6] OF LREAL;
END_VAR
VAR_IN_OUT
	SCP1PCSFRAME : L_UMTP_RobotFrame;
END_VAR
END_METHOD

(* ---- L_MC4P_CLUTCH.pou ---- *)
FUNCTION_BLOCK L_MC4P_CLUTCH
VAR
	XCLUTCHFIRSTCYCLE : BOOL := TRUE;
	XCLUTCHSTARTFORWARD : BOOL;
	XCLUTCHSTARTBACKWARD : BOOL;
	XCLUTCHREADYFORWARD : BOOL;
	XCLUTCHREADYBACKWARD : BOOL;
	SCCHARCLUTCH : ARRAY [0..1] OF L_MC4P_PolyCharacteristics;
	LROLDMAPOS : LREAL;
	ICORRECT : INT;
END_VAR
END_FUNCTION_BLOCK

METHOD CALCPOLY5
VAR_INPUT
	SCCHAR : REFERENCE TO L_MC4P_PolyCharacteristics;
	LRPOS : LREAL;
	PSCNORMSLAVE : POINTER TO L_MC4P_AxisProfile;
END_VAR
END_METHOD

METHOD GENPOLY5ONPOS
VAR_INPUT
	SCACTMASTER : L_MC4P_AxisProfile;
	SCSTARTSLAVE : L_MC4P_AxisProfile;
	SCENDSLAVE : L_MC4P_AxisProfile;
	LRMASTERSTARTPOSITION : LREAL;
	LRMASTERCLUTCHPOSITION : LREAL;
	LRCLUTCHDISTANCE : LREAL;
	LRMASTERSTART : LREAL;
	LRMASTEREND : LREAL;
	LRSLAVEPOSDIFF : LREAL;
	UINUMOFCYCLESMASTER : UINT;
	UINUMOFCYCLESSLAVE : UINT;
	PSCCHARCLUTCH : POINTER TO L_MC4P_PolyCharacteristics;
END_VAR
END_METHOD

METHOD GENERATORCOND
VAR_INPUT
	PSCCHAR : POINTER TO L_MC4P_PolyCharacteristics;
END_VAR
END_METHOD

METHOD PROFILECLUTCHONPOS
VAR_INPUT
	SCACTMASTER : L_MC4P_AxisProfile;
	LRMASTERSTART : LREAL;
	LRMASTEREND : LREAL;
	LRMASTERCLUTCHPOSITION : LREAL;
END_VAR
VAR_OUTPUT
	SCOUTPUTSLAVE : L_MC4P_AxisProfile;
	XCLUTCHDONE : BOOL;
	XERROR : BOOL;
END_VAR
END_METHOD

METHOD RESETCLUTCH
END_METHOD

(* ---- L_MC4P_COORDTRAFO.pou ---- *)
FUNCTION_BLOCK L_MC4P_COORDTRAFO
VAR_INPUT
	COORDTRANSFORM : MC_COORD_REF;
	EROTATIONCONVENTION : L_UMTP_RotationConvention;
END_VAR
VAR_OUTPUT
	T_01 : ARRAY [1..4, 1..4] OF LREAL;
	T_01_FRAME : L_UMTP_RobotFrame;
	T_10 : ARRAY [1..4, 1..4] OF LREAL;
	T_10_FRAME : L_UMTP_RobotFrame;
	T_01_TRACKINGFIXED : ARRAY [1..4, 1..4] OF LREAL;
	T_10_TRACKINGFIXED : ARRAY [1..4, 1..4] OF LREAL;
END_VAR
VAR
	PAXESGROUP : POINTER TO AXES_GROUP_KIN;
	COORDTRANSFORMINT : MC_COORD_REF;
	EROTATIONCONVENTIONINT : L_UMTP_RotationConvention;
	ECOORDSYSINT : L_MC4P_CoordSystem;
END_VAR
END_FUNCTION_BLOCK

METHOD CALCHOMTRAFO
VAR_INPUT
	XUSETRACKINGINITTRAFO : BOOL := FALSE;
	ECOORDSYS : L_MC4P_CoordSystem;
END_VAR
VAR_IN_OUT
	AXESGROUP : AXES_GROUP_KIN;
END_VAR
END_METHOD

METHOD CALCTRAFO_K0_K1
VAR_INPUT
	PALRIN : POINTER TO ARRAY [1..6] OF LREAL;
	PALROUT : POINTER TO ARRAY [1..6] OF LREAL;
	XUSETRACKINGINITTRAFO : BOOL;
END_VAR
END_METHOD

METHOD CALCTRAFO_K1_K0
VAR_INPUT
	PALRIN : POINTER TO ARRAY [1..6] OF LREAL;
	PALROUT : POINTER TO ARRAY [1..6] OF LREAL;
	XUSETRACKINGINITTRAFO : BOOL;
END_VAR
END_METHOD

METHOD ROTATE_K0_K1
VAR_INPUT
	PALRIN : POINTER TO ARRAY [1..6] OF LREAL;
	PALROUT : POINTER TO ARRAY [1..6] OF LREAL;
	XUSETRACKINGINITTRAFO : BOOL;
END_VAR
END_METHOD

METHOD ROTATE_K1_K0
VAR_INPUT
	PALRIN : POINTER TO ARRAY [1..6] OF LREAL;
	PALROUT : POINTER TO ARRAY [1..6] OF LREAL;
	XUSETRACKINGINITTRAFO : BOOL;
END_VAR
END_METHOD

(* ---- L_MC4P_DIFFERENTIALDRIVE2X2.pou ---- *)
FUNCTION_BLOCK L_MC4P_DIFFERENTIALDRIVE2X2 EXTENDS L_MC4P_DifferentialDriveTemplate
VAR_INPUT
	EFIRSTAXIS : IDENT_IN_GROUP_REF;
	ESECONDAXIS : IDENT_IN_GROUP_REF;
	SCDIFFGEARRATIO : L_MC4P_DiffGearFactors2x2;
END_VAR
VAR_OUTPUT
	ALRACSPOSITION : ARRAY [1..2] OF LREAL;
	ALRJCSPOSITION : ARRAY [1..2] OF LREAL;
END_VAR
VAR
	ALRMATRIXFW : ARRAY [1..2, 1..2] OF LREAL;
	ALRMATRIXBW : ARRAY [1..2, 1..2] OF LREAL;
	WAXIS1 : WORD;
	WAXIS2 : WORD;
END_VAR
END_FUNCTION_BLOCK

METHOD BACKWARDTRANSFORMATIONEXTENSION : L_IE1P_Error
VAR_INPUT
	PAXES_POS : POINTER TO ARRAY [1..6] OF LREAL;
	PJOINT_POS : POINTER TO ARRAY [1..6] OF LREAL;
END_VAR
END_METHOD

METHOD CHECKINPUTS : L_IE1P_Error
VAR_IN_OUT
	AXESGROUP : AXES_GROUP_KIN;
END_VAR
END_METHOD

METHOD COPYAXESPOSITIONS
VAR_IN_OUT
	AXESGROUP : AXES_GROUP_KIN;
END_VAR
END_METHOD

METHOD FORWARDTRANSFORMATIONEXTENSION : L_IE1P_Error
VAR_INPUT
	PAXES_POS : POINTER TO ARRAY [1..6] OF LREAL;
	PJOINT_POS : POINTER TO ARRAY [1..6] OF LREAL;
END_VAR
END_METHOD

METHOD GENERALIZEDFORCE_ACS2JCS : L_IE1P_Error
VAR_INPUT
	PAXES_FORCE : POINTER TO ARRAY [1..6] OF LREAL;
	PJOINT_FORCE : POINTER TO ARRAY [1..6] OF LREAL;
END_VAR
END_METHOD

METHOD GENERALIZEDFORCE_JCS2ACS : L_IE1P_Error
VAR_INPUT
	PAXES_FORCE : POINTER TO ARRAY [1..6] OF LREAL;
	PJOINT_FORCE : POINTER TO ARRAY [1..6] OF LREAL;
END_VAR
END_METHOD

METHOD INITIALIZE
END_METHOD

METHOD RESETOUTPUTS
END_METHOD

(* ---- L_MC4P_DIFFERENTIALDRIVE3X3.pou ---- *)
FUNCTION_BLOCK L_MC4P_DIFFERENTIALDRIVE3X3 EXTENDS L_MC4P_DifferentialDriveTemplate
VAR_INPUT
	EFIRSTAXIS : IDENT_IN_GROUP_REF;
	ESECONDAXIS : IDENT_IN_GROUP_REF;
	ETHIRDAXIS : IDENT_IN_GROUP_REF;
	SCDIFFGEARRATIO : L_MC4P_DiffGearFactors3x3;
END_VAR
VAR_OUTPUT
	ALRACSPOSITION : ARRAY [1..3] OF LREAL;
	ALRJCSPOSITION : ARRAY [1..3] OF LREAL;
END_VAR
VAR
	ALRMATRIXFW : ARRAY [1..3, 1..3] OF LREAL;
	ALRMATRIXBW : ARRAY [1..3, 1..3] OF LREAL;
	WAXIS1 : WORD;
	WAXIS2 : WORD;
	WAXIS3 : WORD;
END_VAR
END_FUNCTION_BLOCK

METHOD BACKWARDTRANSFORMATIONEXTENSION : L_IE1P_Error
VAR_INPUT
	PAXES_POS : POINTER TO ARRAY [1..6] OF LREAL;
	PJOINT_POS : POINTER TO ARRAY [1..6] OF LREAL;
END_VAR
END_METHOD

METHOD CHECKINPUTS : L_IE1P_Error
VAR_IN_OUT
	AXESGROUP : AXES_GROUP_KIN;
END_VAR
END_METHOD

METHOD COPYAXESPOSITIONS
VAR_IN_OUT
	AXESGROUP : AXES_GROUP_KIN;
END_VAR
END_METHOD

METHOD FORWARDTRANSFORMATIONEXTENSION : L_IE1P_Error
VAR_INPUT
	PAXES_POS : POINTER TO ARRAY [1..6] OF LREAL;
	PJOINT_POS : POINTER TO ARRAY [1..6] OF LREAL;
END_VAR
END_METHOD

METHOD GENERALIZEDFORCE_ACS2JCS : L_IE1P_Error
VAR_INPUT
	PAXES_FORCE : POINTER TO ARRAY [1..6] OF LREAL;
	PJOINT_FORCE : POINTER TO ARRAY [1..6] OF LREAL;
END_VAR
END_METHOD

METHOD GENERALIZEDFORCE_JCS2ACS : L_IE1P_Error
VAR_INPUT
	PAXES_FORCE : POINTER TO ARRAY [1..6] OF LREAL;
	PJOINT_FORCE : POINTER TO ARRAY [1..6] OF LREAL;
END_VAR
END_METHOD

METHOD INITIALIZE
END_METHOD

METHOD RESETOUTPUTS
END_METHOD

(* ---- L_MC4P_DIFFERENTIALDRIVETEMPLATE.pou ---- *)
FUNCTION_BLOCK L_MC4P_DIFFERENTIALDRIVETEMPLATE EXTENDS L_MC4P_TrafoExtensionBase
VAR_INPUT
	XEXECUTE : BOOL;
	XABORT : BOOL;
END_VAR
VAR_OUTPUT
	XDONE : BOOL;
	XBUSY : BOOL;
	XCOMMANDABORTED : BOOL;
	XERROR : BOOL;
	EERRORID : L_IE1P_Error;
END_VAR
VAR
	XEXECUTEOLD : BOOL;
	XABORTOLD : BOOL;
	EERRORID_TMP : L_IE1P_Error;
	XRESETOUTPUT : BOOL := FALSE;
	XMODULO : BOOL := FALSE;
	XWAITFORDISABLED : BOOL;
END_VAR
END_FUNCTION_BLOCK

METHOD CHECKINPUTS : L_IE1P_Error
VAR_IN_OUT
	AXESGROUP : AXES_GROUP_KIN;
END_VAR
END_METHOD

METHOD COPYAXESPOSITIONS
VAR_IN_OUT
	AXESGROUP : AXES_GROUP_KIN;
END_VAR
END_METHOD

METHOD INITIALIZE
END_METHOD

METHOD MAIN
VAR_IN_OUT
	AXESGROUP : AXES_GROUP_KIN;
END_VAR
END_METHOD

METHOD RESETOUTPUTS
END_METHOD

(* ---- L_MC4P_DYNAMICPAR_AG_KIN.pou ---- *)
FUNCTION_BLOCK L_MC4P_DYNAMICPAR_AG_KIN
VAR_INPUT
	ALRCOULOMBFRICTION : ARRAY [1..6] OF LREAL;
	ALRVISCOSEFRICTION : ARRAY [1..6] OF LREAL;
	ALRGRAVITATIONVECTOR : ARRAY [1..3] OF LREAL := [0, 0, -9.81];
END_VAR
VAR
	GETFRICTIONLOCATION : L_MC4P_PreControlFrictionLocation;
	GETTOOLINERTIA : ARRAY [1..3, 1..3] OF LREAL;
	GETTOOLMASS : LREAL;
END_VAR
END_FUNCTION_BLOCK

METHOD GETDYNAMICPAR : L_IE1P_Error
VAR_IN_OUT
	AXESGROUP : AXES_GROUP_KIN;
	ALRDYNAMICPAR : ARRAY [1..L_MC4P_Constants.uimaxNbrOfDynamicPar] OF LREAL;
END_VAR
END_METHOD

METHOD GETFRICTION : L_IE1P_Error
VAR_IN_OUT
	AXESGROUP : AXES_GROUP_KIN;
	ALRVISCFRIC : ARRAY [1..6] OF LREAL;
	ALRCOULOMBFRIC : ARRAY [1..6] OF LREAL;
END_VAR
END_METHOD

METHOD GETGRAVITATION : L_IE1P_Error
VAR_IN_OUT
	AXESGROUP : AXES_GROUP_KIN;
	ALRGRAVITATION : ARRAY [1..3] OF LREAL;
END_VAR
END_METHOD

METHOD PARAMETERVALID : L_IE1P_Error
VAR_IN_OUT
	AXESGROUP : AXES_GROUP_KIN;
END_VAR
END_METHOD

(* ---- L_MC4P_DYNAMICPARIDENT.pou ---- *)
FUNCTION_BLOCK L_MC4P_DYNAMICPARIDENT EXTENDS L_MC4P_Template_AG_KIN
VAR_INPUT
	XEXECUTE : BOOL;
	ITFDYNAMICPARMIN : L_MC4P_DynamicPar;
	ITFDYNAMICPARMAX : L_MC4P_DynamicPar;
	XUSEAXESLIMITS : BOOL;
	ALRMINPOS : ARRAY [1..6] OF LREAL;
	ALRMAXPOS : ARRAY [1..6] OF LREAL;
	ALRMAXVEL : ARRAY [1..6] OF LREAL;
	ALRMAXACC : ARRAY [1..6] OF LREAL;
END_VAR
VAR_OUTPUT
	XDONE : BOOL;
	XBUSY : BOOL;
	XACTIVE : BOOL;
	XCOMMANDABORTED : BOOL;
	XERROR : BOOL;
	EERRORID : L_IE1P_Error;
	LRCONVERGENCE : LREAL;
END_VAR
VAR
	SCTRAFOINFO : L_MC4P_TrafoInfo;
	SCERROR : L_MC4P_ErrorStruct;
	ALRDYNAMICPARIDENT : ARRAY [1..L_MC4P_Constants.uimaxNbrOfDynamicPar] OF LREAL;
	ALRVISCFRICIDENT : ARRAY [1..6] OF LREAL;
	ALRCOULOMBFRICIDENT : ARRAY [1..6] OF LREAL;
	ALRGRAVITATIONIDENT : ARRAY [1..3] OF LREAL;
	WADAPTSTEP : WORD;
	WADAPTPARAMSTEP : WORD := 20;
	XACTVALUESFORIDENT : BOOL := TRUE;
	EIDENTMODE_INT : L_MC4P_IdentMode := L_MC4P_IdentMode.CompleteModel;
	XIDENTCURRENTMOVEMENT_INT : BOOL := FALSE;
	WSTEP : WORD := 0;
	WSTEPOLD : WORD := 0;
	XFIRSTCYCLEINSTEP : BOOL;
	XEXECUTEOLD : BOOL;
	XRESETOUTPUTS : BOOL;
	PASCFOURIERPARAM : POINTER TO ARRAY [1..6] OF L_MC4P_IdentTrajectoryFourierParam;
	ESPACEOFMOTION : L_MC4P_SpaceOfMotion;
	USINBROFDYNPAR : USINT;
	USIACTNBROFAXES : USINT;
	AUSISIZEOFREGREESIONMATRIX : ARRAY [1..2] OF USINT;
	PLRREGRESSIONMATRIX : POINTER TO LREAL;
	PLRPARAMS : POINTER TO LREAL;
	PLRPARAMSMIN : POINTER TO LREAL;
	PLRPARAMSMAX : POINTER TO LREAL;
	PLRDUMMY : POINTER TO LREAL;
	USIIDENTCYCLE : USINT;
	USIIDENTCYCLEMAX : USINT;
	LRINTERPOLATIONTIME : LREAL := 0.0;
	USIFOURIERCYCLES : USINT := 6;
	LRFOURIERPERIOD : LREAL;
	XLIMITSAVAILABLE : BOOL;
	ALRVISCFRICMIN : ARRAY [1..6] OF LREAL;
	ALRCOULOMBFRICMIN : ARRAY [1..6] OF LREAL;
	ALRDYNAMICPARMIN : ARRAY [1..L_MC4P_Constants.uimaxNbrOfDynamicPar] OF LREAL;
	ALRVISCFRICMAX : ARRAY [1..6] OF LREAL;
	ALRCOULOMBFRICMAX : ARRAY [1..6] OF LREAL;
	ALRDYNAMICPARMAX : ARRAY [1..L_MC4P_Constants.uimaxNbrOfDynamicPar] OF LREAL;
	ALRACSPOSATEXECUTE : ARRAY [1..6] OF LREAL;
	ALRSTARTPOSITION_EXCITATION : ARRAY [1..6] OF LREAL;
	ALRSTARTPOSITION_AXES : ARRAY [1..6] OF LREAL;
	ALRFOURIERPOSITION : ARRAY [1..usiBufferSize] OF ARRAY [1..6] OF LREAL;
	ALRFOURIERVELOCITY : ARRAY [1..usiBufferSize] OF ARRAY [1..6] OF LREAL;
	ALRFOURIERACCELERATION : ARRAY [1..usiBufferSize] OF ARRAY [1..6] OF LREAL;
	ALRFOURIERPOSITION2 : ARRAY [1..usiBufferSize] OF ARRAY [1..6] OF LREAL;
	ALRFOURIERVELOCITY2 : ARRAY [1..usiBufferSize] OF ARRAY [1..6] OF LREAL;
	ALRFOURIERACCELERATION2 : ARRAY [1..usiBufferSize] OF ARRAY [1..6] OF LREAL;
	ALRSETPOSITION : ARRAY [1..6] OF LREAL;
	ALRSETVELOCITY : ARRAY [1..6] OF LREAL;
	ALRSETACCELERATION : ARRAY [1..6] OF LREAL;
	ALRACTPOSITION : ARRAY [1..6] OF LREAL;
	ALRACTVELOCITY : ARRAY [1..6] OF LREAL;
	ALRACTACCELERATION : ARRAY [1..6] OF LREAL;
	ALRACTTORQUEACS : ARRAY [1..6] OF LREAL;
	ALRACTTORQUEJCS : ARRAY [1..6] OF LREAL;
	ALRACTACSPOS : ARRAY [1..6] OF LREAL;
	ALRACTACSVEL : ARRAY [1..6] OF LREAL;
	ALRACTACSACC : ARRAY [1..6] OF LREAL;
	ALREXTTORQUE : ARRAY [1..6] OF LREAL;
	ALRCALCULATEDTORQUEJCS : ARRAY [1..6] OF LREAL;
	USIWRITEIDX : USINT;
	USIWRITEIDXOLD : USINT;
	USIREADIDX : USINT;
	USIBUSDELAY : USINT := 5;
	LRFADINGRATIO : LREAL := 0.5;
	LRFADINGFAKTOR : LREAL;
	LRDFADINGFAKTOR : LREAL;
	LRDDFADINGFAKTOR : LREAL;
	RLS1 : L_UMTP_RLS;
	IDX : UINT;
	IDXAXISOFFSET : UINT;
	ALRMINPOS_INT : ARRAY [1..6] OF LREAL;
	ALRMAXPOS_INT : ARRAY [1..6] OF LREAL;
	ALRMAXVEL_INT : ARRAY [1..6] OF LREAL;
	ALRMAXACC_INT : ARRAY [1..6] OF LREAL;
	LRMAXCARTVEL : LREAL;
	LRMAXCARTACC : LREAL;
	XDIFFERENTIALDRIVE1ACTIVE : BOOL;
	PACTTRAFOEXTENSION1 : POINTER TO L_MC4P_TrafoExtensionBase;
	LRACTVALUEFILTERTIME : LREAL := 0.01;
	LRFILTERTIMEFACTOR : LREAL := 50;
	APOSPT1 : ARRAY [1..6] OF L_USPP_PT1Filter;
	AVELPT1 : ARRAY [1..6] OF L_USPP_PT1Filter;
	AACCPT1 : ARRAY [1..6] OF L_USPP_PT1Filter;
	ATORQUEPT1 : ARRAY [1..6] OF L_USPP_PT1Filter;
	AGOF : ARRAY [1..6] OF L_UMTP_GoodnessOfFit;
	LRCONVERGENCEWARNINGLEVEL : LREAL := 0.8;
	LRCONVERGENCEERRORLEVEL : LREAL := 0.6;
	LRCONVERGENCECOLOR : LREAL;
	LRMINOR : LREAL;
	LRMINORLIM : LREAL := 0.8;
	LRVERIFICATIONBLENDPERC : LREAL := 25.0;
	USIBUFFERSIZE : USINT := 8;
	GETFRICTIONLOCATION : L_MC4P_PreControlFrictionLocation;
	GETTOOLINERTIA : ARRAY [1..3, 1..3] OF LREAL;
	GETTOOLMASS : LREAL;
	LOWEROVERRIDELIMIT : LREAL;
	LRTRANSITIONPARAMETER2 : LREAL;
END_VAR
END_FUNCTION_BLOCK

METHOD ADAPTFOURIERPARAM : BOOL
VAR_IN_OUT
	AXESGROUP : AXES_GROUP_KIN;
END_VAR
END_METHOD

METHOD AXESVALUESTOFOURIERCOORDSYSTEM
VAR_IN_OUT
	AXESGROUP : AXES_GROUP_KIN;
	ALRFOURIERPOSITION : ARRAY [1..6] OF LREAL;
	ALRFOURIERVELOCITY : ARRAY [1..6] OF LREAL;
	ALRFOURIERACCELERATION : ARRAY [1..6] OF LREAL;
	ALRSETPOSITION : ARRAY [1..6] OF LREAL;
	ALRSETVELOCITY : ARRAY [1..6] OF LREAL;
	ALRSETACCELERATION : ARRAY [1..6] OF LREAL;
END_VAR
END_METHOD

METHOD CALCFADINGFUNCTION
VAR_IN_OUT
	AXESGROUP : AXES_GROUP_KIN;
END_VAR
END_METHOD

METHOD EVALUATEFOURIERAXIS
VAR_INPUT
	LRT : LREAL;
	LROVERRIDE : LREAL;
	IDXAXIS : UINT;
END_VAR
VAR_OUTPUT
	LRPOS_EXCITATION : LREAL;
	LRVEL_EXCITATION : LREAL;
	LRACC_EXCITATION : LREAL;
	LRPOS_AXES : LREAL;
	LRVEL_AXES : LREAL;
	LRACC_AXES : LREAL;
END_VAR
END_METHOD

METHOD GOTOIDLE
VAR_IN_OUT
	AXESGROUP : AXES_GROUP_KIN;
END_VAR
END_METHOD

METHOD IDENTALLOWED : BOOL
VAR_IN_OUT
	AXESGROUP : AXES_GROUP_KIN;
END_VAR
END_METHOD

METHOD INITVERIFICATION : BOOL
VAR_IN_OUT
	AXESGROUP : AXES_GROUP_KIN;
END_VAR
END_METHOD

METHOD READINPUTS
VAR_IN_OUT
	AXESGROUP : AXES_GROUP_KIN;
END_VAR
END_METHOD

METHOD RESETOUTPUTS
END_METHOD

METHOD TRANSFORMFOURIERPARAMS_AXES2EXCITATION
VAR_IN_OUT
	AXESGROUP : AXES_GROUP_KIN;
END_VAR
END_METHOD

METHOD TRANSFORMFOURIERPARAMS_EXCITATION2AXES
VAR_IN_OUT
	AXESGROUP : AXES_GROUP_KIN;
END_VAR
END_METHOD

METHOD VERIFY
VAR_IN_OUT
	AXESGROUP : AXES_GROUP_KIN;
END_VAR
END_METHOD

METHOD FB_SETSCERROR : BOOL
END_METHOD

METHOD GETDYNAMICPAR : L_IE1P_Error
VAR_IN_OUT
	AXESGROUP : AXES_GROUP_KIN;
	ALRDYNAMICPAR : ARRAY [1..L_MC4P_Constants.uimaxNbrOfDynamicPar] OF LREAL;
END_VAR
END_METHOD

METHOD GETFRICTION : L_IE1P_Error
VAR_IN_OUT
	AXESGROUP : AXES_GROUP_KIN;
	ALRVISCFRIC : ARRAY [1..6] OF LREAL;
	ALRCOULOMBFRIC : ARRAY [1..6] OF LREAL;
END_VAR
END_METHOD

METHOD GETGRAVITATION : L_IE1P_Error
VAR_IN_OUT
	AXESGROUP : AXES_GROUP_KIN;
	ALRGRAVITATION : ARRAY [1..3] OF LREAL;
END_VAR
END_METHOD

METHOD PARAMETERVALID : L_IE1P_Error
VAR_IN_OUT
	AXESGROUP : AXES_GROUP_KIN;
END_VAR
END_METHOD

(* ---- L_MC4P_EXTDYNAMICSBASE.pou ---- *)
FUNCTION_BLOCK L_MC4P_EXTDYNAMICSBASE EXTENDS L_MC4P_Template_AG_KIN
VAR_INPUT
	XENABLE : BOOL;
END_VAR
VAR_OUTPUT
	XBUSY : BOOL;
	XERROR : BOOL;
	EERRORID : L_IE1P.L_IE1P_Error;
END_VAR
VAR
	XENABLEOLD : BOOL;
	XWAITFORDISABLED : BOOL;
	XERRORWRITEITF : BOOL;
	XERRORREADINPUTS : BOOL;
END_VAR
END_FUNCTION_BLOCK

METHOD CALCEXTACSTORQUE
VAR_INPUT
	ALRACSPOS : ARRAY [1..6] OF LREAL;
	ALRACSVEL : ARRAY [1..6] OF LREAL;
	ALRACSACC : ARRAY [1..6] OF LREAL;
END_VAR
VAR_OUTPUT
	ALREXTTORQUE : ARRAY [1..6] OF LREAL;
END_VAR
END_METHOD

METHOD READINPUTS
VAR_IN_OUT
	AXESGROUP : AXES_GROUP_KIN;
END_VAR
END_METHOD

METHOD RESETOUTPUTS
VAR_IN_OUT
	AXESGROUP : AXES_GROUP_KIN;
END_VAR
END_METHOD

(* ---- L_MC4P_FILTERORCOMBINE.pou ---- *)
FUNCTION_BLOCK L_MC4P_FILTERORCOMBINE EXTENDS L_USPP_Filter
VAR_INPUT
	ORFAST : REFERENCE TO L_MC4P_FilterORFast;
	ORLEGACY : REFERENCE TO L_MC4P_FilterORLegacy;
END_VAR
VAR_OUTPUT
	EOVRTYPEUSED : L_MC4P_OVRType := L_MC4P_OVRType.OvrTypePoly;
END_VAR
END_FUNCTION_BLOCK

METHOD CYCLICACTION
VAR_INPUT
	ITFTIMINGCONTROLLER : L_UBUP.L_UBUP_ITimingController;
END_VAR
VAR_OUTPUT
	XCOMPLETE : BOOL;
	XABORT : BOOL;
	IERRORID : INT;
END_VAR
END_METHOD

METHOD STARTACTION
VAR_OUTPUT
	XCOMPLETE : BOOL;
	IERRORID : INT;
END_VAR
END_METHOD

METHOD FB_INIT : BOOL
VAR_INPUT
	BINITRETAINS : BOOL;
	BINCOPYCODE : BOOL;
END_VAR
END_METHOD

METHOD INIT
END_METHOD

METHOD LOGIK
END_METHOD

(* ---- L_MC4P_FILTERORFAST.pou ---- *)
FUNCTION_BLOCK L_MC4P_FILTERORFAST EXTENDS L_USPP_Filter
VAR_INPUT
	LRDAMP : LREAL := 0.95;
END_VAR
VAR_OUTPUT
	XLIMITSVIOLATED : BOOL;
END_VAR
VAR
	_AXESGROUP : REFERENCE TO AXES_GROUP_KIN;
	_IDYNLIMITPROVIDER : L_MC4P_IDynLimitProvider;
	_PLISTELEMENTACTIVE : POINTER TO L_MC4P_ListElement;
	_V_ACS : REFERENCE TO ARRAY [1..6] OF LREAL;
	_A_ACS : REFERENCE TO ARRAY [1..6] OF LREAL;
	_V_WCS : REFERENCE TO ARRAY [4..6] OF LREAL;
	_A_WCS : REFERENCE TO ARRAY [4..6] OF LREAL;
	_V_AUX : REFERENCE TO ARRAY [1..6] OF LREAL;
	_A_AUX : REFERENCE TO ARRAY [1..6] OF LREAL;
	_PATHPOS : REFERENCE TO LREAL;
	_PASSED_PATHPOS : REFERENCE TO LREAL;
	_PATHVEL : REFERENCE TO LREAL;
	_PATHACC : REFERENCE TO LREAL;
	_LRACTTIMEOR : REFERENCE TO LREAL;
	_LRACTTIMEDOR : REFERENCE TO LREAL;
	_XCONNECTED : BOOL := FALSE;
	_REFPROFILES : REFERENCE TO L_MC4P_ListElementDataProfiles;
	_REFPATH : REFERENCE TO L_MC4P_PathData;
	_LROVRREQUEST : LREAL;
	_BNOMOTION : BOOL;
	_VEL_MAX : ARRAY [1..6] OF LREAL;
	_ACC_MAX : ARRAY [1..6] OF LREAL;
	_ACC_MIN : ARRAY [1..6] OF LREAL;
	_VEL_AUX_MAX : ARRAY [1..6] OF LREAL;
	_ACC_AUX_MAX : ARRAY [1..6] OF LREAL;
	_ACC_AUX_MIN : ARRAY [1..6] OF LREAL;
	_VEL_MAX_PATH : LREAL;
	_ACC_MAX_PATH : LREAL;
	_ACC_MIN_PATH : LREAL;
	_BUP : BOOL;
	_LRRESULT : LREAL;
	_LRINVCYCLETIME : LREAL := -1;
	_LRCYCLETIMEOLD : LREAL := -1;
	_SCSP : L_MC4P_CyclicData;
	_DTMAX : LREAL := 0.0001;
	_ORFAST_EPS : LREAL := 0.0001;
END_VAR
END_FUNCTION_BLOCK

METHOD CONNECTTOINTERPOLATOR
VAR_INPUT
	AXESGROUP : REFERENCE TO AXES_GROUP_KIN;
END_VAR
END_METHOD

METHOD SETACTIVELISTELEMENT
VAR_INPUT
	PLISTELEMENT : POINTER TO L_MC4P_ListElement;
END_VAR
END_METHOD

METHOD CYCLICACTION
VAR_INPUT
	ITFTIMINGCONTROLLER : L_UBUP.L_UBUP_ITimingController;
END_VAR
VAR_OUTPUT
	XCOMPLETE : BOOL;
	XABORT : BOOL;
	IERRORID : INT;
END_VAR
END_METHOD

METHOD STARTACTION
VAR_OUTPUT
	XCOMPLETE : BOOL;
	IERRORID : INT;
END_VAR
END_METHOD

METHOD FIRSTDERIV
VAR_INPUT
	PLRY : POINTER TO LREAL;
	PLRDY : POINTER TO LREAL;
	UDIDIM : UDINT;
	LRT : LREAL;
END_VAR
END_METHOD

METHOD FB_INIT : BOOL
VAR_INPUT
	BINITRETAINS : BOOL;
	BINCOPYCODE : BOOL;
END_VAR
END_METHOD

METHOD GETAUXAXESLIMITS
END_METHOD

METHOD GETMAINAXESLIMITS
END_METHOD

METHOD GETPATHLIMITS
END_METHOD

METHOD GETREALAXESLIMITS
END_METHOD

METHOD GETROTAXESLIMITS
END_METHOD

METHOD INTEGRATEOVR : LREAL
END_METHOD

METHOD OVRDERIV_COMPLETE : LREAL
VAR_INPUT
	Y : LREAL;
	T : LREAL;
END_VAR
END_METHOD

METHOD OVRDERIV_AUX : LREAL
VAR_INPUT
	Y : LREAL;
	T : LREAL;
END_VAR
END_METHOD

METHOD OVRDERIV_LIMITTOAXES : LREAL
VAR_INPUT
	Y : LREAL;
	T : LREAL;
END_VAR
END_METHOD

METHOD OVRDERIV_PTP : LREAL
VAR_INPUT
	Y : LREAL;
	T : LREAL;
END_VAR
END_METHOD

METHOD OVRDERIV_PATH : LREAL
VAR_INPUT
	Y : LREAL;
	T : LREAL;
END_VAR
END_METHOD

METHOD OVRDERIV_ROT : LREAL
VAR_INPUT
	Y : LREAL;
	T : LREAL;
END_VAR
END_METHOD

(* ---- L_MC4P_FILTERORLEGACY.pou ---- *)
FUNCTION_BLOCK L_MC4P_FILTERORLEGACY EXTENDS L_USPP_Filter
VAR_INPUT
	PAXESGROUP : POINTER TO AXES_GROUP_KIN;
	LRTIMEOR_FADETIME : LREAL;
END_VAR
VAR
	LRSETTIMEOR : LREAL;
	LRSETTIMEOR_OLD : LREAL;
	LRACTTIMEOR : REFERENCE TO LREAL;
	LRACTTIMEOR_OLD : LREAL;
	LRACTTIMEDOR : REFERENCE TO LREAL;
	ALRORCOEFFS : ARRAY [0..3] OF LREAL;
	ALRORCOEFFS_INT : ARRAY [0..3] OF LREAL;
	LRTIMEORIPOTIME : LREAL;
	LRTIMEORDECTIME : LREAL;
	LRTIMEOR_FADETIME_OLD : LREAL;
	IORLOCKCOUNTER : INT;
	IORLOCKCOUNTERMAX : INT := 2;
	LRTIMEORSETDIFF : LREAL;
	LRTIMEORDECTIME_INT : LREAL;
	XNEWCOEFFICIENTS : BOOL := FALSE;
END_VAR
END_FUNCTION_BLOCK

METHOD FORCEACTUALOVR : L_IE1P_Error
VAR_INPUT
	LROVRACTUAL : LREAL;
END_VAR
END_METHOD

METHOD CYCLICACTION
VAR_INPUT
	ITFTIMINGCONTROLLER : L_UBUP.L_UBUP_ITimingController;
END_VAR
VAR_OUTPUT
	XCOMPLETE : BOOL;
	XABORT : BOOL;
	IERRORID : INT;
END_VAR
END_METHOD

METHOD STARTACTION
VAR_OUTPUT
	XCOMPLETE : BOOL;
	IERRORID : INT;
END_VAR
END_METHOD

METHOD FB_INIT : BOOL
VAR_INPUT
	BINITRETAINS : BOOL;
	BINCOPYCODE : BOOL;
END_VAR
END_METHOD

(* ---- L_MC4P_FUNIDMANAGER.pou ---- *)
FUNCTION_BLOCK L_MC4P_FUNIDMANAGER
VAR_OUTPUT
	DIFUNID : DINT;
	DIACTFUNID : DINT;
	DIBUSYFUNID : DINT;
	DIABORTFUNID : DINT;
	XWAITINGFORPROFILEPREPAXESGROUP : BOOL := FALSE;
	XWAITINGFORPROFILEPREPAXESGROUPOLD : BOOL := FALSE;
	XMOVEFBWAITINGFOREMPTYLIST : BOOL;
END_VAR
VAR
	DILOOKAHEADFUNID : DINT;
	XDONTKILLFUNID : BOOL;
	XISBEINGABORTED : BOOL;
END_VAR
END_FUNCTION_BLOCK

METHOD FORWARDBUSYID
VAR_IN_OUT
	PATHLIST : L_MC4P_PathDataList;
	SCTRACKINGHANDSHAKE : L_MC4P_TrackingHandshake;
END_VAR
END_METHOD

METHOD KEEPFUNIDTHISCYCLE
END_METHOD

METHOD REGISTERFUNCTION : DINT
END_METHOD

METHOD RESETIDS
END_METHOD

METHOD SETABORTINGFUNID
VAR_INPUT
	DIABORTFUNID : DINT;
END_VAR
END_METHOD

METHOD SETFUNIDSTOVALUE
VAR_INPUT
	DIID : DINT;
END_VAR
END_METHOD

METHOD SETMOVEFBWAITINGFOREMPTYLIST
VAR_INPUT
	XMOVEFBWAITINGFOREMPTYLIST : BOOL;
END_VAR
END_METHOD

(* ---- L_MC4P_GEOOBJECTBASE.pou ---- *)
FUNCTION_BLOCK L_MC4P_GEOOBJECTBASE
VAR_INPUT
	PINST : POINTER TO L_MC4P_GeoObjectInst;
	PLISTELEMENT : POINTER TO L_MC4P_ListElement;
END_VAR
VAR_OUTPUT
	NSTATE : DINT;
	XISREADY : BOOL := FALSE;
	XERROR : BOOL := FALSE;
	SCERROR : L_MC4P_ErrorStruct;
END_VAR
VAR
	XHASZEROLENGTH : BOOL := FALSE;
	FINALPATHCOORDINATE : LREAL;
	LENGTH : LREAL;
	MAXBENDING : LREAL;
	STARTPATHCOORDINATE : LREAL;
	STATESIZE : UDINT;
END_VAR
END_FUNCTION_BLOCK

METHOD BENDING : BOOL
VAR_INPUT
	LRPATHPOS : LREAL;
END_VAR
VAR_OUTPUT
	LRBENDING : LREAL;
	SCERROR : L_MC4P_ErrorStruct;
END_VAR
END_METHOD

METHOD CALCMAXBEND : BOOL
END_METHOD

METHOD CALCNORMPOS : BOOL
VAR_INPUT
	LRPATHCOORD : LREAL;
	REFERROR : REFERENCE TO L_MC4P_ErrorStruct;
END_VAR
VAR_OUTPUT
	LRPATHCOORD_NORMED : LREAL;
END_VAR
END_METHOD

METHOD COPYFROM : BOOL
VAR_INPUT
	REFGEOOBJECT : REFERENCE TO L_MC4P_GeoObjectBase;
END_VAR
END_METHOD

METHOD CUT : BOOL
VAR_INPUT
	LRS0 : LREAL;
	LRS1 : LREAL;
END_VAR
VAR_OUTPUT
	SCERROR : L_MC4P_ErrorStruct;
END_VAR
END_METHOD

METHOD EXPANDLISTELEMENT : BOOL
VAR_OUTPUT
	SCERROR : L_MC4P_ErrorStruct;
END_VAR
END_METHOD

METHOD FINALIZE : BOOL
END_METHOD

METHOD GETFINALSETPOINTDATA : BOOL
VAR_OUTPUT
	SCERROR : L_MC4P_ErrorStruct;
END_VAR
VAR_IN_OUT
	SCSP : L_MC4P_CyclicData;
END_VAR
END_METHOD

METHOD GETINSTANCE : REFERENCE TO L_MC4P_GeoObjectInst
END_METHOD

METHOD GETLISTELEMENTDATA : REFERENCE TO L_MC4P_ListElementData
END_METHOD

METHOD GETSETPOINDATA : BOOL
VAR_OUTPUT
	SCERROR : L_MC4P_ErrorStruct;
END_VAR
VAR_IN_OUT
	SCSP : L_MC4P_CyclicData;
END_VAR
END_METHOD

METHOD GETSETPOINDATA_NORMED : BOOL
VAR_INPUT
	BPOS : BOOL;
	BVEL : BOOL;
	BACC : BOOL;
END_VAR
VAR_IN_OUT
	SCSP : L_MC4P_CyclicData;
	SCERROR : L_MC4P_ErrorStruct;
END_VAR
END_METHOD

METHOD MAPTOPATHCOORDINATE : BOOL
VAR_OUTPUT
	SCERROR : L_MC4P_ErrorStruct;
END_VAR
END_METHOD

METHOD UPDATEBOUNDS : BOOL
VAR_OUTPUT
	SCERROR : L_MC4P_ErrorStruct;
END_VAR
END_METHOD

METHOD WRITETOFILE : BOOL
VAR_INPUT
	SPATH : STRING;
END_VAR
END_METHOD

METHOD RESET : BOOL
VAR_INPUT
	PBYSTATE : POINTER TO BYTE;
	UDISIZE : UDINT;
END_VAR
VAR_OUTPUT
	SCERROR : L_MC4P_ErrorStruct;
END_VAR
END_METHOD

METHOD STORESTATE : BOOL
VAR_INPUT
	PBYSTATE : POINTER TO BYTE;
	UDISIZE : UDINT;
END_VAR
VAR_OUTPUT
	SCERROR : L_MC4P_ErrorStruct;
END_VAR
END_METHOD

(* ---- L_MC4P_GEOOBJECTCIRCLE.pou ---- *)
FUNCTION_BLOCK L_MC4P_GEOOBJECTCIRCLE EXTENDS L_MC4P_GeoObjectBase
END_FUNCTION_BLOCK

METHOD BENDING : BOOL
VAR_INPUT
	LRPATHPOS : LREAL;
END_VAR
VAR_OUTPUT
	LRBENDING : LREAL;
	SCERROR : L_MC4P_ErrorStruct;
END_VAR
END_METHOD

METHOD EXPANDLISTELEMENT : BOOL
VAR_OUTPUT
	SCERROR : L_MC4P_ErrorStruct;
END_VAR
END_METHOD

METHOD GETSETPOINDATA_NORMED : BOOL
VAR_INPUT
	BPOS : BOOL;
	BVEL : BOOL;
	BACC : BOOL;
END_VAR
VAR_IN_OUT
	SCSP : L_MC4P_CyclicData;
	SCERROR : L_MC4P_ErrorStruct;
END_VAR
END_METHOD

METHOD MAPTOPATHCOORDINATE : BOOL
VAR_OUTPUT
	SCERROR : L_MC4P_ErrorStruct;
END_VAR
END_METHOD

METHOD UPDATEBOUNDS : BOOL
VAR_OUTPUT
	SCERROR : L_MC4P_ErrorStruct;
END_VAR
END_METHOD

(* ---- L_MC4P_GEOOBJECTCUBICSPLINE.pou ---- *)
FUNCTION_BLOCK L_MC4P_GEOOBJECTCUBICSPLINE EXTENDS L_MC4P_GeoObjectBase
END_FUNCTION_BLOCK

METHOD CALCCUBICSPLINE
VAR_INPUT
	REFCUBICSPLINE : REFERENCE TO L_MC4P_CubicSplineData;
	REFTARGETPOS : REFERENCE TO ARRAY [1..6] OF LREAL;
	REFERROR : REFERENCE TO L_MC4P_ErrorStruct;
END_VAR
END_METHOD

METHOD CALCSPLINEBENDINGMAX : LREAL
VAR_INPUT
	REFCUBICSPLINE : REFERENCE TO L_MC4P_CubicSplineData;
END_VAR
END_METHOD

METHOD EXPANDLISTELEMENT : BOOL
VAR_OUTPUT
	SCERROR : L_MC4P_ErrorStruct;
END_VAR
END_METHOD

METHOD GETSETPOINDATA_NORMED : BOOL
VAR_INPUT
	BPOS : BOOL;
	BVEL : BOOL;
	BACC : BOOL;
END_VAR
VAR_IN_OUT
	SCSP : L_MC4P_CyclicData;
	SCERROR : L_MC4P_ErrorStruct;
END_VAR
END_METHOD

METHOD MAPTOPATHCOORDINATE : BOOL
VAR_OUTPUT
	SCERROR : L_MC4P_ErrorStruct;
END_VAR
END_METHOD

METHOD UPDATEBOUNDS : BOOL
VAR_OUTPUT
	SCERROR : L_MC4P_ErrorStruct;
END_VAR
END_METHOD

(* ---- L_MC4P_GEOOBJECTELLIPSE.pou ---- *)
FUNCTION_BLOCK L_MC4P_GEOOBJECTELLIPSE EXTENDS L_MC4P_GeoObjectBase
END_FUNCTION_BLOCK

METHOD CALCNORMPOS : BOOL
VAR_INPUT
	LRPATHCOORD : LREAL;
	REFERROR : REFERENCE TO L_MC4P_ErrorStruct;
END_VAR
VAR_OUTPUT
	LRPATHCOORD_NORMED : LREAL;
END_VAR
END_METHOD

METHOD EXPANDLISTELEMENT : BOOL
VAR_OUTPUT
	SCERROR : L_MC4P_ErrorStruct;
END_VAR
END_METHOD

METHOD GETSETPOINDATA_NORMED : BOOL
VAR_INPUT
	BPOS : BOOL;
	BVEL : BOOL;
	BACC : BOOL;
END_VAR
VAR_IN_OUT
	SCSP : L_MC4P_CyclicData;
	SCERROR : L_MC4P_ErrorStruct;
END_VAR
END_METHOD

METHOD MAPPARABEL
VAR_IN_OUT
	SCELLIPSE : L_MC4P_EllipseData;
	ALRLENGTH : ARRAY [1..L_MC4P_Constants.LengthVec_idxmax] OF LREAL;
END_VAR
END_METHOD

METHOD MAPTOPATHCOORDINATE : BOOL
VAR_OUTPUT
	SCERROR : L_MC4P_ErrorStruct;
END_VAR
END_METHOD

METHOD UPDATEBOUNDS : BOOL
VAR_OUTPUT
	SCERROR : L_MC4P_ErrorStruct;
END_VAR
END_METHOD

(* ---- L_MC4P_GEOOBJECTNURBS.pou ---- *)
FUNCTION_BLOCK L_MC4P_GEOOBJECTNURBS EXTENDS L_MC4P_GeoObjectBase
END_FUNCTION_BLOCK

(* ---- L_MC4P_GEOOBJECTPOLYNOM.pou ---- *)
FUNCTION_BLOCK L_MC4P_GEOOBJECTPOLYNOM EXTENDS L_MC4P_GeoObjectBase
END_FUNCTION_BLOCK

METHOD BENDING : BOOL
VAR_INPUT
	LRPATHPOS : LREAL;
END_VAR
VAR_OUTPUT
	LRBENDING : LREAL;
	SCERROR : L_MC4P_ErrorStruct;
END_VAR
END_METHOD

METHOD CALC1STDERIVATIVE : ARRAY [1..3] OF LREAL
VAR_INPUT
	PATHKOEFF : REFERENCE TO ARRAY [1..3, 1..6] OF LREAL;
	S_NORM : LREAL;
END_VAR
END_METHOD

METHOD CALC2NDDERIVATIVE : ARRAY [1..3] OF LREAL
VAR_INPUT
	PATHKOEFF : REFERENCE TO ARRAY [1..3, 1..6] OF LREAL;
	S_NORM : LREAL;
END_VAR
END_METHOD

METHOD CALCMAXBENDING : LREAL
VAR_INPUT
	ESEGMENTTYPE : L_MC4P_SegmentType;
	PATHKOEFF : ARRAY [1..3, 1..6] OF LREAL;
END_VAR
END_METHOD

METHOD CALCPATHKOEFF : ARRAY [1..3, 1..6] OF LREAL
VAR_INPUT
	ESEGMENTTYPE : L_MC4P_SegmentType;
	X0 : ARRAY [1..6] OF LREAL;
	X1 : ARRAY [1..6] OF LREAL;
	X0STRICH : ARRAY [1..3] OF LREAL;
	X1STRICH : ARRAY [1..3] OF LREAL;
	X02STRICH : ARRAY [1..3] OF LREAL;
	X12STRICH : ARRAY [1..3] OF LREAL;
END_VAR
END_METHOD

METHOD CALCSEGMENTLENGTH : LREAL
VAR_INPUT
	IDXMAX : INT;
	ESEGMENTTYPE : L_MC4P_SegmentType;
	PATHKOEFF : ARRAY [1..3, 1..6] OF LREAL;
END_VAR
END_METHOD

METHOD CALCSEGMENTLENGTHVEC
VAR_INPUT
	ESEGMENTTYPE : L_MC4P_SegmentType;
	PATHKOEFF : REFERENCE TO ARRAY [1..3, 1..6] OF LREAL;
END_VAR
VAR_IN_OUT
	LENGTH : ARRAY [1..L_MC4P_Constants.LengthVec_idxmax] OF LREAL;
END_VAR
END_METHOD

METHOD EXPANDLISTELEMENT : BOOL
VAR_OUTPUT
	SCERROR : L_MC4P_ErrorStruct;
END_VAR
END_METHOD

METHOD EXPANDLISTELEMENT_P1 : BOOL
VAR_OUTPUT
	SCERROR : L_MC4P_ErrorStruct;
END_VAR
END_METHOD

METHOD EXPANDLISTELEMENT_P5 : BOOL
VAR_OUTPUT
	SCERROR : L_MC4P_ErrorStruct;
END_VAR
END_METHOD

METHOD GETSETPOINDATA_NORMED : BOOL
VAR_INPUT
	BPOS : BOOL;
	BVEL : BOOL;
	BACC : BOOL;
END_VAR
VAR_IN_OUT
	SCSP : L_MC4P_CyclicData;
	SCERROR : L_MC4P_ErrorStruct;
END_VAR
END_METHOD

METHOD MAPTOPATHCOORDINATE : BOOL
VAR_OUTPUT
	SCERROR : L_MC4P_ErrorStruct;
END_VAR
END_METHOD

METHOD UPDATEBOUNDS : BOOL
VAR_OUTPUT
	SCERROR : L_MC4P_ErrorStruct;
END_VAR
END_METHOD

(* ---- L_MC4P_GEOOBJECTPROVIDER.pou ---- *)
FUNCTION_BLOCK L_MC4P_GEOOBJECTPROVIDER
VAR_INPUT
	PLISTELEMENT : POINTER TO L_MC4P_ListElement;
END_VAR
VAR_OUTPUT
	NSTATE : DINT;
	XERROR : BOOL := FALSE;
	SCERROR : L_MC4P_ErrorStruct;
END_VAR
VAR
	FBPOLYNOM : L_MC4P_GeoObjectPolynom;
	FBCIRCLE : L_MC4P_GeoObjectCircle;
	FBCUBICSPLINE : L_MC4P_GeoObjectCubicSpline;
	FBELLIPSE : L_MC4P_GeoObjectEllipse;
	FBPTP : L_MC4P_GeoObjectPTP;
	SCINST : L_MC4P_GeoObjectInst;
	ITFGEOOBJECT : L_MC4P_IGeoObject;
	GEOOBJECT : L_MC4P_IGeoObject;
END_VAR
END_FUNCTION_BLOCK

METHOD COPYFROM : BOOL
VAR_INPUT
	PNEW : POINTER TO L_MC4P_ListElement;
	PSOURCE : POINTER TO L_MC4P_ListElement;
END_VAR
VAR_OUTPUT
	SCERROR : L_MC4P_ErrorStruct;
END_VAR
END_METHOD

METHOD FINALIZE : BOOL
END_METHOD

(* ---- L_MC4P_GEOOBJECTPTP.pou ---- *)
FUNCTION_BLOCK L_MC4P_GEOOBJECTPTP EXTENDS L_MC4P_GeoObjectBase
END_FUNCTION_BLOCK

METHOD EXPANDLISTELEMENT : BOOL
VAR_OUTPUT
	SCERROR : L_MC4P_ErrorStruct;
END_VAR
END_METHOD

METHOD GETSETPOINDATA_NORMED : BOOL
VAR_INPUT
	BPOS : BOOL;
	BVEL : BOOL;
	BACC : BOOL;
END_VAR
VAR_IN_OUT
	SCSP : L_MC4P_CyclicData;
	SCERROR : L_MC4P_ErrorStruct;
END_VAR
END_METHOD

METHOD UPDATEBOUNDS : BOOL
VAR_OUTPUT
	SCERROR : L_MC4P_ErrorStruct;
END_VAR
END_METHOD

(* ---- L_MC4P_GETACTIVETOOL.pou ---- *)
FUNCTION_BLOCK L_MC4P_GETACTIVETOOL EXTENDS L_MC4P_Template_AG_KIN
VAR_INPUT
	XEXECUTE : BOOL;
END_VAR
VAR_OUTPUT
	XDONE : BOOL;
	XBUSY : BOOL;
	XERROR : BOOL;
	EERRORID : L_IE1P_Error := L_IE1P_Error.NoError;
	ETOOLSYSTEM : L_MC4P_ToolSystem;
	SCTOOLPARAMETER : L_MC4P_TOOL_REF;
END_VAR
VAR
	XEXECUTEOLD : BOOL;
	XRESETOUTPUT : BOOL;
	ALRVISUTOOLPARAMETER : ARRAY [1..8] OF LREAL;
	PTOOL : POINTER TO L_MC4P_ToolTrafo;
END_VAR
END_FUNCTION_BLOCK

(* ---- L_MC4P_GROUPDIGITALSWITCHHANDLER.pou ---- *)
FUNCTION_BLOCK L_MC4P_GROUPDIGITALSWITCHHANDLER EXTENDS L_MC4P_Template_AG_KIN
VAR_INPUT
	XENABLE : BOOL;
	XRESETSWITCHES : BOOL;
END_VAR
VAR_OUTPUT
	XVALID : BOOL;
	XBUSY : BOOL;
	XERROR : BOOL;
	EERRORID : L_IE1P_Error;
	DWDIGITALSWITCHES : DWORD;
END_VAR
VAR
	ADWDIGITALSWITCHES : ARRAY [1..cwNbrOfdwDigSwitches] OF DWORD;
	LRPASSEDLENGTHOFSEGMENTID : LREAL;
	LRPASSEDTIMEOFSEGMENTID : LREAL;
	_MODEL : L_UBUP_BehaviourModel_LCon;
	XRESETSWITCHESOLD : BOOL;
	RSCSWITCHINGFUN : REFERENCE TO L_MC4P_SwitchingFunctionData;
	ALRSWITCHPARAMSORTED : ARRAY [1..L_MC4P_Constants.gciMaxNumParallelSwitchingFun] OF LREAL;
	XPOSRELATED : BOOL;
	ISWITCHIDXVISU : INT := 1;
	WVISUIDX : WORD := 1;
	CWNBROFDWDIGSWITCHES : WORD := 1024;
	IDXMAX : DINT;
	IDXMIN : DINT;
END_VAR
END_FUNCTION_BLOCK

METHOD ANALYZEANDSORTDATA : BOOL
VAR_INPUT
	PLISTELEMENT : POINTER TO L_MC4P_ListElement;
END_VAR
END_METHOD

METHOD GETDIGITALSWITCH : BOOL
VAR_INPUT
	WDIGITALSWITCH : WORD;
END_VAR
END_METHOD

METHOD RESET : BOOL
END_METHOD

METHOD SETDIGITALSWITCH : BOOL
VAR_INPUT
	WDIGITALSWITCH : WORD;
	XVALUE : BOOL;
END_VAR
END_METHOD

METHOD SETEVALUATEDFLAG : BOOL
VAR_INPUT
	PLISTELEMENT : POINTER TO L_MC4P_ListElement;
	IDX : INT;
END_VAR
END_METHOD

METHOD SPLITINDEX : BOOL
VAR_INPUT
	WSWITCHIDX : WORD;
END_VAR
VAR_OUTPUT
	WARRIDX : WORD;
	WBITIDX : WORD;
END_VAR
END_METHOD

METHOD CYCLICIPOCALL : BOOL
VAR_INPUT
	PLISTELEMENT : POINTER TO L_MC4P_ListElement;
	RSCCYCLICDATA : REFERENCE TO L_MC4P_CyclicData;
END_VAR
END_METHOD

METHOD FINALIZESEGMENT : BOOL
VAR_INPUT
	PLISTELEMENTACT : POINTER TO L_MC4P_ListElement;
	PLISTELEMENTNEXT : POINTER TO L_MC4P_ListElement;
END_VAR
END_METHOD

METHOD CYCLICACTION
VAR_INPUT
	ITFTIMINGCONTROLLER : L_UBUP.L_UBUP_ITimingController;
END_VAR
VAR_OUTPUT
	XCOMPLETE : BOOL;
	XABORT : BOOL;
	IERRORID : INT;
END_VAR
END_METHOD

METHOD FINALIZEACTION
VAR_INPUT
	XABORTPROPOSED : BOOL;
	IERRORIDPROPOSED : INT;
END_VAR
VAR_OUTPUT
	XCOMPLETE : BOOL;
	XABORT : BOOL;
	IERRORID : INT;
END_VAR
END_METHOD

METHOD RESETACTION
VAR_OUTPUT
	XCOMPLETE : BOOL;
END_VAR
END_METHOD

METHOD STARTACTION
VAR_OUTPUT
	XCOMPLETE : BOOL;
	IERRORID : INT;
END_VAR
END_METHOD

METHOD EXCHANGE : BOOL
VAR_INPUT
	IDX1 : DINT;
	IDX2 : DINT;
END_VAR
END_METHOD

METHOD GETVALUE : LREAL
VAR_INPUT
	IDX : DINT;
END_VAR
END_METHOD

(* ---- L_MC4P_GROUPHOME_INTERNAL.pou ---- *)
FUNCTION_BLOCK L_MC4P_GROUPHOME_INTERNAL EXTENDS L_UBUP_PoolInstance
VAR_INPUT
	EXECUTE : BOOL;
END_VAR
VAR_OUTPUT
	DONE : BOOL;
	BUSY : BOOL;
	ACTIVE : BOOL;
	COMMANDABORTED : BOOL;
	ERROR : BOOL;
	ERRORID : L_IE1P_Error;
	AXISDONE : ARRAY [1..12] OF BOOL;
END_VAR
VAR
	COORDSYSTEM : L_MC4P_CoordSystem := L_MC4P_CoordSystem.ACS;
	AMC_HOME : ARRAY [1..12] OF L_MC1P_Home_Internal;
	AMC_HOME_FBBASE : ARRAY [1..12] OF L_MC1P_Template;
	XRESETOUTPUT : BOOL;
	XEXECUTEOLD : BOOL;
	XVALIDAXISSTATES : BOOL;
	IDX : WORD;
	EACTHOMINGORDER : L_MC4P_HomingOrder := L_MC4P_HomingOrder.NoHoming;
	AXAXESHOMED : ARRAY [1..12] OF BOOL;
	ALRPOSITION_INT : ARRAY [1..12] OF LREAL;
	AEHOMINGORDER_INT : ARRAY [1..12] OF L_MC4P_HomingOrder := [12(0)];
	ECOORDSYSTEM_INT : L_MC4P_CoordSystem;
	ASCEXTPARAMETER_INT : ARRAY [1..12] OF L_MC1P_HomeParameter;
	AXUSEEXTPARAMETER_INT : ARRAY [1..12] OF BOOL;
	ASCEXTTP_INT : ARRAY [1..12] OF MC_TRIGGER_REF;
	CLASSID : DINT;
END_VAR
END_FUNCTION_BLOCK

METHOD MAIN
VAR_IN_OUT
	AXESGROUP : AXES_GROUP_KIN;
	FBBASE : L_MC4P_Template_AG_KIN;
	POSITION : ARRAY [1..12] OF LREAL;
	HOMINGORDER : ARRAY [1..12] OF L_MC4P_HomingOrder;
	HOMEABSSWITCH : ARRAY [1..12] OF BOOL;
	USEEXTPARAMETER : ARRAY [1..12] OF BOOL;
	EXTPARAMETER : ARRAY [1..12] OF L_MC1P_HomeParameter;
	EXTTP : ARRAY [1..12] OF MC_TRIGGER_REF;
END_VAR
END_METHOD

METHOD RESETOUTPUTS
END_METHOD

METHOD SETAXISMC_HOME_ACS : BOOL
VAR_IN_OUT
	AXESGROUP : AXES_GROUP_KIN;
	FBBASE : L_MC4P_Template_AG_KIN;
	HOMEABSSWITCH : ARRAY [1..12] OF BOOL;
END_VAR
END_METHOD

METHOD SETNEXTHOMESTEP
END_METHOD

METHOD GET_EERRORID : L_IE1P_Error
END_METHOD

METHOD GET_XACTIVE : BOOL
END_METHOD

METHOD GET_XBUSY : BOOL
END_METHOD

METHOD GET_XCOMMANDABORTED : BOOL
END_METHOD

METHOD GET_XDONE : BOOL
END_METHOD

METHOD GET_XINITIAL : BOOL
END_METHOD

METHOD FREE : BOOL
END_METHOD

(* ---- L_MC4P_GROUPMANUALMODE.pou ---- *)
FUNCTION_BLOCK L_MC4P_GROUPMANUALMODE EXTENDS L_MC4P_Template_AG_KIN
VAR_INPUT
	ALRSETPOSDIST : ARRAY [1..12] OF LREAL;
	SCPAR : L_MC4P_GroupManualMode_Parameter;
	ECOORDSYSTEM : L_MC4P_CoordSystem;
	AXJOGPOS : ARRAY [1..12] OF BOOL;
	AXJOGNEG : ARRAY [1..12] OF BOOL;
	AXMOVEABSEXECUTE : ARRAY [1..12] OF BOOL;
	AXMOVERELEXECUTE : ARRAY [1..12] OF BOOL;
END_VAR
VAR_OUTPUT
	XINTERNALCONTROLACTIVE : BOOL;
	XBUSY : BOOL;
	XDONE : BOOL;
	XERROR : BOOL;
	EERRORID : L_IE1P_Error;
	EMANUALMODE : L_MC4P_ManualMode := L_MC4P_ManualMode.Standby;
END_VAR
VAR
	MANMODE : L_MC4P_GroupManualMode_Internal;
END_VAR
END_FUNCTION_BLOCK

(* ---- L_MC4P_GROUPMANUALMODE_INTERNAL.pou ---- *)
FUNCTION_BLOCK L_MC4P_GROUPMANUALMODE_INTERNAL EXTENDS L_UBUP_PoolInstance
VAR_INPUT
	ALRSETPOSDIST : ARRAY [1..12] OF LREAL;
	SCPAR : L_MC4P_GroupManualMode_Parameter;
	ECOORDSYSTEM : L_MC4P_CoordSystem;
	AXJOGPOS : ARRAY [1..12] OF BOOL;
	AXJOGNEG : ARRAY [1..12] OF BOOL;
	AXMOVEABSEXECUTE : ARRAY [1..12] OF BOOL;
	AXMOVERELEXECUTE : ARRAY [1..12] OF BOOL;
	XISV2 : BOOL := FALSE;
END_VAR
VAR_OUTPUT
	XINTERNALCONTROLACTIVE : BOOL;
	XBUSY : BOOL;
	XDONE : BOOL;
	XERROR : BOOL;
	EERRORID : L_IE1P_Error;
	EMANUALMODE : L_MC4P_ManualMode := L_MC4P_ManualMode.Standby;
END_VAR
VAR
	AXMOVEABSEXECUTEEDGE : ARRAY [1..12] OF BOOL;
	AXMOVERELEXECUTEEDGE : ARRAY [1..12] OF BOOL;
	ECOORDSYSTEM_INT : L_MC4P_CoordSystem := L_MC4P_CoordSystem.MCS;
	XDOSTATEMACHINE : BOOL;
	XCHANGETOSTANDBY : BOOL := FALSE;
	XJOGGING : BOOL;
	XMOVEABSEDGE : BOOL;
	XMOVERELEDGE : BOOL;
	XMOVEABS : BOOL;
	XMOVEREL : BOOL;
	AMANUALJOG : ARRAY [1..12] OF L_MC1P_ManualJog_Internal;
	AMANUALJOG_FBBASE : ARRAY [1..12] OF L_MC1P.L_MC1P_Template;
	AMC_MOVERELATIVE : ARRAY [1..12] OF L_MC1P_MoveRelative_Internal;
	AMC_MOVERELATIVE_FBBASE : ARRAY [1..12] OF L_MC1P.L_MC1P_Template;
	AMC_MOVEABSOLUTE : ARRAY [1..12] OF L_MC1P_MoveAbsolute_Inernal;
	AMC_MOVEABSOLUTE_FBBASE : ARRAY [1..12] OF L_MC1P.L_MC1P_Template;
	EMANUALMODEOLD : L_MC4P_ManualMode := L_MC4P_ManualMode.Standby;
	ECOORDSYSTEMOLD : L_MC4P_CoordSystem;
	AXMOVEABSEXECUTEOLD : ARRAY [1..12] OF BOOL;
	AXMOVERELEXECUTEOLD : ARRAY [1..12] OF BOOL;
	XMOTIONACTIVE : BOOL := FALSE;
	APG : ARRAY [1..6] OF L_MC1P.L_MC1P_PosProfiler;
	ASCPROFILEPARAMETER : ARRAY [1..6] OF L_MC1P_ProfileParameter;
	PCOORDTRAFO : POINTER TO L_MC4P_CoordTrafo;
	COORDTRAFO_INT : L_MC4P_CoordTrafo;
	ALRPCSSETPOSATEXECUTE : ARRAY [1..6] OF LREAL;
	PLRDUMMY : POINTER TO LREAL;
	ALRPCSSETPOS_EXT : ARRAY [1..6] OF LREAL;
	ALRWCSSETPOS_EXT : ARRAY [1..6] OF LREAL;
	CLASSID : DINT;
END_VAR
END_FUNCTION_BLOCK

METHOD MAIN
VAR_IN_OUT
	AXESGROUP : AXES_GROUP_KIN;
	FBBASE : L_MC4P_Template_AG_KIN;
END_VAR
END_METHOD

METHOD GET_EERRORID : L_IE1P_Error
END_METHOD

METHOD GET_XACTIVE : BOOL
END_METHOD

METHOD GET_XBUSY : BOOL
END_METHOD

METHOD GET_XCOMMANDABORTED : BOOL
END_METHOD

METHOD GET_XDONE : BOOL
END_METHOD

METHOD GET_XINITIAL : BOOL
END_METHOD

METHOD FREE : BOOL
END_METHOD

METHOD CHECKPCSMCS : BOOL
END_METHOD

METHOD ENTRYSTANDBYSTATE
VAR_IN_OUT
	AXESGROUP : AXES_GROUP_KIN;
	FBBASE : L_MC4P_Template_AG_KIN;
END_VAR
END_METHOD

METHOD EXITMOVESTATE
VAR_IN_OUT
	AXESGROUP : AXES_GROUP_KIN;
	FBBASE : L_MC4P_Template_AG_KIN;
END_VAR
END_METHOD

METHOD GETTCSPOSINPCSMCS
VAR_INPUT
	EROTATIONCONVENTIONPCS : L_UMTP_RotationConvention;
END_VAR
VAR_IN_OUT
	AXESGROUP : AXES_GROUP_KIN;
	ALRPCSSETPOS : ARRAY [1..6] OF LREAL;
END_VAR
END_METHOD

METHOD ISMOTIONALLOWED
VAR_IN_OUT
	AXESGROUP : AXES_GROUP_KIN;
	FBBASE : L_MC4P_Template_AG_KIN;
	SCPAR : L_MC4P_GroupManualMode_Parameter;
	ECOORDSYSTEM : L_MC4P_CoordSystem;
	AXJOGPOS : ARRAY [1..12] OF BOOL;
	AXJOGNEG : ARRAY [1..12] OF BOOL;
	AXMOVEABSEXECUTE : ARRAY [1..12] OF BOOL;
	AXMOVERELEXECUTE : ARRAY [1..12] OF BOOL;
END_VAR
END_METHOD

METHOD JOGAXISREF
VAR_INPUT
	XWCS : BOOL;
	XACS : BOOL;
	XAUX : BOOL;
END_VAR
VAR_IN_OUT
	AXESGROUP : AXES_GROUP_KIN;
	FBBASE : L_MC4P_Template_AG_KIN;
	SCPAR : L_MC4P_GroupManualMode_Parameter;
	AXJOGPOS : ARRAY [1..12] OF BOOL;
	AXJOGNEG : ARRAY [1..12] OF BOOL;
END_VAR
END_METHOD

METHOD JOGPCSMCS
VAR_IN_OUT
	AXESGROUP : AXES_GROUP_KIN;
	FBBASE : L_MC4P_Template_AG_KIN;
	SCPAR : L_MC4P_GroupManualMode_Parameter;
	AXJOGPOS : ARRAY [1..12] OF BOOL;
	AXJOGNEG : ARRAY [1..12] OF BOOL;
END_VAR
END_METHOD

METHOD MOVEABSAXISREF
VAR_INPUT
	XWCS : BOOL;
	XACS : BOOL;
	XAUX : BOOL;
END_VAR
VAR_IN_OUT
	AXESGROUP : AXES_GROUP_KIN;
	FBBASE : L_MC4P_Template_AG_KIN;
	ALRSETPOSDIST : ARRAY [1..12] OF LREAL;
	SCPAR : L_MC4P_GroupManualMode_Parameter;
	AXMOVEABSEXECUTE : ARRAY [1..12] OF BOOL;
END_VAR
END_METHOD

METHOD MOVEABSPCSMCS
VAR_IN_OUT
	AXESGROUP : AXES_GROUP_KIN;
	FBBASE : L_MC4P_Template_AG_KIN;
	ALRSETPOSDIST : ARRAY [1..12] OF LREAL;
	SCPAR : L_MC4P_GroupManualMode_Parameter;
	AXMOVEABSEXECUTE : ARRAY [1..12] OF BOOL;
END_VAR
END_METHOD

METHOD MOVERELAXISREF
VAR_INPUT
	XWCS : BOOL;
	XACS : BOOL;
	XAUX : BOOL;
END_VAR
VAR_IN_OUT
	AXESGROUP : AXES_GROUP_KIN;
	FBBASE : L_MC4P_Template_AG_KIN;
	ALRSETPOSDIST : ARRAY [1..12] OF LREAL;
	SCPAR : L_MC4P_GroupManualMode_Parameter;
	AXMOVERELEXECUTE : ARRAY [1..12] OF BOOL;
END_VAR
END_METHOD

METHOD MOVERELPCSMCS
VAR_IN_OUT
	AXESGROUP : AXES_GROUP_KIN;
	FBBASE : L_MC4P_Template_AG_KIN;
	ALRSETPOSDIST : ARRAY [1..12] OF LREAL;
	SCPAR : L_MC4P_GroupManualMode_Parameter;
	AXMOVERELEXECUTE : ARRAY [1..12] OF BOOL;
END_VAR
END_METHOD

METHOD RESETMOTIONQUERY
END_METHOD

METHOD WRITEPCSMCSPOS2AXES
VAR_INPUT
	EROTATIONCONVENTIONPCS : L_UMTP_RotationConvention;
	XRELATIVE : BOOL;
END_VAR
VAR_IN_OUT
	AXESGROUP : AXES_GROUP_KIN;
	FBBASE : L_MC4P_Template_AG_KIN;
	ALRPCSSETPOS : ARRAY [1..6] OF LREAL;
	ALRPCSSETVEL : ARRAY [1..6] OF LREAL;
END_VAR
END_METHOD

METHOD CALL_AXISREFPARM
VAR_INPUT
	AXESGROUP : REFERENCE TO AXES_GROUP_KIN;
	LRVELOCITY : REFERENCE TO LREAL;
	LRACCELERATION : REFERENCE TO LREAL;
	LRDECELERATION : REFERENCE TO LREAL;
	LRJERK : REFERENCE TO LREAL;
	AXIS_IDX_LOCAL : WORD;
END_VAR
END_METHOD

METHOD CALL_PCSMCSPARM
VAR_INPUT
	AXESGROUP : REFERENCE TO AXES_GROUP_KIN;
	ALRPCSSETPOS : REFERENCE TO ARRAY [1..6] OF LREAL;
	IDX_LOCAL : WORD;
END_VAR
END_METHOD

(* ---- L_MC4P_GROUPPOWER.pou ---- *)
FUNCTION_BLOCK L_MC4P_GROUPPOWER EXTENDS L_MC4P_Template_AG_REF
VAR_INPUT
	XENABLE : BOOL;
	AEAXISENABLE : ARRAY [1..12] OF L_MC4P_AxisEnableMode := [12(L_MC4P_AxisEnableMode.EnablePosNeg)];
END_VAR
VAR_OUTPUT
	XSTATUS : BOOL;
	XVALID : BOOL;
	XERROR : BOOL;
	EERRORID : L_IE1P_Error;
END_VAR
VAR
	AMC_POWER : ARRAY [1..12] OF MC_Power;
	XENABLEOLD : BOOL;
	IDX : WORD;
	IDX_PLUSSIX : WORD;
	XAXISEXTENABLED : BOOL := FALSE;
	XERRORINTERN : BOOL := FALSE;
	EERRORIDINTERN : L_IE1P_Error;
	XAXISERROR : BOOL := FALSE;
END_VAR
END_FUNCTION_BLOCK

(* ---- L_MC4P_GROUPREADACTUALPOSITION_INTERNAL.pou ---- *)
FUNCTION_BLOCK L_MC4P_GROUPREADACTUALPOSITION_INTERNAL EXTENDS L_UBUP_Instance
VAR_INPUT
	ENABLE : BOOL;
	COORDSYSTEM : L_MC4P_CoordSystem;
END_VAR
VAR_OUTPUT
	VALID : BOOL;
	BUSY : BOOL;
	ERROR : BOOL;
	ERRORID : L_IE1P_Error;
END_VAR
VAR
	IDX : WORD;
	XENABLEOLD : BOOL;
	PCOORDTRAFO : POINTER TO L_MC4P_CoordTrafo;
	ALRPOSITIONTMP : ARRAY [1..6] OF LREAL;
	CLASSID : DINT;
END_VAR
END_FUNCTION_BLOCK

METHOD MAIN
VAR_INPUT
	XUSESETVALUES : BOOL;
END_VAR
VAR_IN_OUT
	AXESGROUP : AXES_GROUP_KIN;
	FBBASE : L_MC4P_Template_AG_KIN;
	POSITION : ARRAY [1..12] OF LREAL;
END_VAR
END_METHOD

(* ---- L_MC4P_GROUPREADACTUALVELOCITY_INTERNAL.pou ---- *)
FUNCTION_BLOCK L_MC4P_GROUPREADACTUALVELOCITY_INTERNAL EXTENDS L_UBUP_Instance
VAR_INPUT
	ENABLE : BOOL;
	COORDSYSTEM : L_MC4P_CoordSystem;
END_VAR
VAR_OUTPUT
	VALID : BOOL;
	BUSY : BOOL;
	ERROR : BOOL;
	ERRORID : L_IE1P_Error;
END_VAR
VAR
	IDX : WORD;
	XENABLEOLD : BOOL;
	ALRVELOCITYTMP1 : ARRAY [1..6] OF LREAL;
	ALRVELOCITYTMP2 : ARRAY [1..6] OF LREAL;
	ALRPOSITIONTMP : ARRAY [1..6] OF LREAL;
	PCOORDTRAFO : POINTER TO L_MC4P_CoordTrafo;
	ALRPOSVEKPCS2TCS : ARRAY [1..3] OF LREAL;
	ROT_MAT : ARRAY [1..3, 1..3] OF LREAL;
	T4 : LREAL;
	T5 : LREAL;
	T7 : LREAL;
	CLASSID : DINT;
END_VAR
END_FUNCTION_BLOCK

METHOD MAIN
VAR_INPUT
	XUSESETVALUES : BOOL;
END_VAR
VAR_IN_OUT
	AXESGROUP : AXES_GROUP_KIN;
	FBBASE : L_MC4P_Template_AG_KIN;
	VELOCITY : ARRAY [1..12] OF LREAL;
	PATHVELOCITY : LREAL;
END_VAR
END_METHOD

(* ---- L_MC4P_GROUPREADSTATUS_INTERNAL.pou ---- *)
FUNCTION_BLOCK L_MC4P_GROUPREADSTATUS_INTERNAL EXTENDS L_UBUP_PoolInstance
VAR_INPUT
	ENABLE : BOOL;
END_VAR
VAR_OUTPUT
	VALID : BOOL;
	BUSY : BOOL;
	ERROR : BOOL;
	ERRORID : L_IE1P_Error;
	GROUPMOVING : BOOL;
	GROUPHOMING : BOOL;
	GROUPERRORSTOP : BOOL;
	GROUPSTANDBY : BOOL;
	GROUPSTOPPING : BOOL;
	GROUPDISABLED : BOOL;
	CONSTANTVELOCITY : BOOL;
	ACCELERATING : BOOL;
	DECELERATING : BOOL;
	INPOSITION : BOOL;
	STANDSTILL : BOOL;
END_VAR
VAR
	XENABLEOLD : BOOL;
	IDX : INT;
	CLASSID : DINT;
END_VAR
END_FUNCTION_BLOCK

METHOD MAIN
VAR_IN_OUT
	AXESGROUP : AXES_GROUP_KIN;
	FBBASE : L_MC4P_Template_AG_KIN;
END_VAR
END_METHOD

(* ---- L_MC4P_GROUPRESET_INTERNAL.pou ---- *)
FUNCTION_BLOCK L_MC4P_GROUPRESET_INTERNAL EXTENDS L_UBUP_Instance
VAR_INPUT
	EXECUTE : BOOL;
END_VAR
VAR_OUTPUT
	DONE : BOOL;
	BUSY : BOOL;
	ERROR : BOOL;
	ERRORID : L_IE1P_Error;
END_VAR
VAR
	ARESET : ARRAY [1..18] OF MC_Reset;
	PAXESGROUP : POINTER TO AXES_GROUP_KIN;
	XEXECUTEOLD : BOOL;
	PWTMP : POINTER TO WORD;
	IDX : INT;
	XRESETPOSSIBLE : BOOL;
	XRESETOUTPUT : BOOL;
	DWRESETCYCLECOUNTERSTART : DWORD;
	XNOERRORACTIVE : BOOL;
	XERRORSTOPDONE : BOOL;
	XAXESGROUPINERROR : BOOL;
	XAXISINERROR : BOOL;
	XWAITFORRESETEVENT : BOOL;
	DWMAXTIMEOUT : DWORD;
	CLASSID : DINT;
END_VAR
END_FUNCTION_BLOCK

METHOD MAIN
VAR_IN_OUT
	AXESGROUP : AXES_GROUP_REF;
	FBBASE : L_MC4P_Template_ForAG;
END_VAR
END_METHOD

METHOD REQUESTINTERFACE : BOOL
VAR_INPUT
	ID : DINT;
	PITFUNKNOWN : POINTER TO L_UBUP_IUnknown;
END_VAR
END_METHOD

(* ---- L_MC4P_GROUPSETOVERRIDE.pou ---- *)
FUNCTION_BLOCK L_MC4P_GROUPSETOVERRIDE EXTENDS L_MC4P_Template_AG_KIN
VAR_INPUT
	XENABLE : BOOL;
	LROVERRIDE : LREAL := 1.0;
	LRFADINGTIME : LREAL := 2.5;
END_VAR
VAR_OUTPUT
	XENABLED : BOOL;
	XBUSY : BOOL;
	XERROR : BOOL;
	EERRORID : L_IE1P_Error := L_IE1P_Error.NoError;
END_VAR
VAR
	GROUPSETOVERRIDE : L_MC4P_GroupSetOverride_Internal;
END_VAR
END_FUNCTION_BLOCK

(* ---- L_MC4P_GROUPSETOVERRIDE_INTERNAL.pou ---- *)
FUNCTION_BLOCK L_MC4P_GROUPSETOVERRIDE_INTERNAL EXTENDS L_UBUP_PoolInstance
VAR_INPUT
	XENABLE : BOOL;
	LROVERRIDE : LREAL := 1.0;
	LRFADINGTIME : LREAL := 2.5;
END_VAR
VAR_OUTPUT
	XENABLED : BOOL;
	XBUSY : BOOL;
	XERROR : BOOL;
	EERRORID : L_IE1P_Error := L_IE1P_Error.NoError;
END_VAR
VAR
	XENABLEOLD : BOOL;
	CLASSID : DINT;
END_VAR
END_FUNCTION_BLOCK

METHOD MAIN
VAR_IN_OUT
	AXESGROUP : AXES_GROUP_KIN;
	FBBASE : L_MC4P_Template_AG_KIN;
END_VAR
END_METHOD

METHOD REQUESTINTERFACE : BOOL
VAR_INPUT
	ID : DINT;
	PITFUNKNOWN : POINTER TO L_UBUP_IUnknown;
END_VAR
END_METHOD

(* ---- L_MC4P_GROUPSETPOSITION_INTERNAL.pou ---- *)
FUNCTION_BLOCK L_MC4P_GROUPSETPOSITION_INTERNAL EXTENDS L_UBUP_PoolInstance
VAR_INPUT
	EXECUTE : BOOL;
	RELATIVE : BOOL := FALSE;
END_VAR
VAR_OUTPUT
	DONE : BOOL;
	BUSY : BOOL;
	ACTIVE : BOOL;
	ERROR : BOOL;
	ERRORID : L_IE1P_Error;
END_VAR
VAR
	COORDSYSTEM : L_MC4P_CoordSystem := L_MC4P_CoordSystem.ACS;
	XRESETOUTPUT : BOOL;
	AMC_SETPOSITION : ARRAY [1..12] OF L_MC1P.MC_SetPosition;
	IDX : WORD;
	XEXECUTEOLD : BOOL;
	CLASSID : DINT;
END_VAR
END_FUNCTION_BLOCK

METHOD MAIN
VAR_IN_OUT
	AXESGROUP : AXES_GROUP_KIN;
	FBBASE : L_MC4P_Template_AG_KIN;
	POSITION : ARRAY [1..12] OF LREAL;
END_VAR
END_METHOD

METHOD REQUESTINTERFACE : BOOL
VAR_INPUT
	ID : DINT;
	PITFUNKNOWN : POINTER TO L_UBUP_IUnknown;
END_VAR
END_METHOD

(* ---- L_MC4P_GROUPSTOP_INTERNAL.pou ---- *)
FUNCTION_BLOCK L_MC4P_GROUPSTOP_INTERNAL EXTENDS L_MC4P_CalcStopProfiles
VAR_INPUT
	EXECUTE : BOOL;
	DECELERATION : LREAL;
	JERK : LREAL;
END_VAR
VAR_OUTPUT
	DONE : BOOL;
	BUSY : BOOL;
	ACTIVE : BOOL;
	COMMANDABORTED : BOOL;
	ERROR : BOOL;
	ERRORID : L_IE1P_Error;
END_VAR
VAR
	_ITFOWNER : L_UBUP.L_UBUP_IFBPool;
	_XWHANDLE : __XWORD;
	_XOCCUPIED : BOOL;
	LRINPUTJERK : LREAL;
	LRINPUTDECELERATION : LREAL;
	AMC_STOP : ARRAY [1..18] OF L_MC1P.L_MC1P_Stop_Internal;
	AMC_STOP_FBBASE : ARRAY [1..18] OF L_MC1P.L_MC1P_Template;
	IDX : WORD;
	XEXECUTEOLD : BOOL;
	XRESETOUTPUT : BOOL;
	XDONEINTERN : BOOL;
	XDONEOLD : BOOL;
	XERRORINTERN : BOOL;
	EERRORIDINTERN : L_IE1P_Error;
	DWINTERNALID : DWORD;
	XSTOPPROFILESCALCULATED : BOOL;
	_DWOBJID : DWORD;
	CLASSID : DINT;
	INSTANCEPTR : POINTER TO BYTE;
	OBJECTID : DWORD;
	OCCUPIED : BOOL;
END_VAR
END_FUNCTION_BLOCK

METHOD GROUPSTOPACS
VAR_IN_OUT
	AXESGROUP : AXES_GROUP_KIN;
	FBBASE : L_MC4P_Template_AG_KIN;
END_VAR
END_METHOD

METHOD GROUPSTOPMCS
VAR_IN_OUT
	AXESGROUP : AXES_GROUP_KIN;
	FBBASE : L_MC4P_Template_AG_KIN;
END_VAR
END_METHOD

METHOD MAIN
VAR_IN_OUT
	AXESGROUP : AXES_GROUP_KIN;
	FBBASE : L_MC4P_Template_AG_KIN;
END_VAR
END_METHOD

METHOD RESETOUTPUTS
VAR_IN_OUT
	AXESGROUP : AXES_GROUP_KIN;
END_VAR
END_METHOD

METHOD GET_EERRORID : L_IE1P_Error
END_METHOD

METHOD GET_XACTIVE : BOOL
END_METHOD

METHOD GET_XBUSY : BOOL
END_METHOD

METHOD GET_XCOMMANDABORTED : BOOL
END_METHOD

METHOD GET_XDONE : BOOL
END_METHOD

METHOD GET_XINITIAL : BOOL
END_METHOD

METHOD FREE : BOOL
END_METHOD

METHOD OCCUPY : BOOL
VAR_INPUT
	ITFOWNER : L_UBUP.L_UBUP_IFBPool;
	XWHANDLE : __XWORD;
END_VAR
END_METHOD

METHOD REQUESTINTERFACE : BOOL
VAR_INPUT
	ID : DINT;
	PITFUNKNOWN : POINTER TO L_UBUP_IUnknown;
END_VAR
END_METHOD

METHOD FB_INIT : BOOL
VAR_INPUT
	BINITRETAINS : BOOL;
	BINCOPYCODE : BOOL;
END_VAR
END_METHOD

(* ---- L_MC4P_GROUPTORQUEPRECONTROL.pou ---- *)
FUNCTION_BLOCK L_MC4P_GROUPTORQUEPRECONTROL EXTENDS L_MC4P_Template_AG_KIN
VAR_INPUT
	XENABLE : BOOL;
	XUSEAXESGROUPPARAM : BOOL := FALSE;
	XWRITETOPARAMETER : BOOL := FALSE;
	LRTORQUEOVERRIDE : LREAL := 0;
	LRTORQUELIMITFACTOR : LREAL := 1;
	ALRTORQUERATELIMIT : ARRAY [1..6] OF LREAL := [6(0.0)];
	LRLOADMASS : LREAL;
	ITFDYNAMICPAR : L_MC4P_DynamicPar;
END_VAR
VAR_OUTPUT
	XVALID : BOOL;
	XBUSY : BOOL;
	XERROR : BOOL;
	EERRORID : L_IE1P_Error;
	ALRSETTORQUEOUT : ARRAY [1..6] OF LREAL;
	ALRACTTORQUE : ARRAY [1..6] OF LREAL;
END_VAR
VAR
	LICHANDLING : L_IMHP_LLMHandling;
	IDX : INT;
	IDX2 : WORD;
	XENABLEOLD : BOOL;
	XWRITETOPARAMETEROLD : BOOL;
	ALRTORQUELIMITS : ARRAY [1..6] OF LREAL;
	ALRTORQUEDELTACYCLE : ARRAY [1..6] OF LREAL := [6(0.0)];
	XUSEFILTEREDVALUES : BOOL := TRUE;
	XSETVALUEFILTERACTIVE : BOOL;
	EBEHAVEONERRORSTOP : L_MC4P_ErrorStopBehaviour := L_MC4P_ErrorStopBehaviour.SetTorqueToZero;
	ALRGRAVITATION : ARRAY [1..3] OF LREAL;
	ALRCOULOMBFRIC : ARRAY [1..6] OF LREAL;
	ALRVISCFRIC : ARRAY [1..6] OF LREAL;
	ALRDYNAMICPAR : ARRAY [1..L_MC4P_Constants.uimaxNbrOfDynamicPar] OF LREAL;
	EERRORTMP : L_IE1P_Error;
	ALRTOOLINERTIA : ARRAY [1..3, 1..3] OF LREAL;
	ALRLOADINERTIA : ARRAY [1..3, 1..3] OF LREAL;
	BEHAVEONERRORSTOP : L_MC4P_ErrorStopBehaviour;
	USEFILTEREDVALUES : BOOL;
END_VAR
END_FUNCTION_BLOCK

(* ---- L_MC4P_GROUPWAITTIME.pou ---- *)
FUNCTION_BLOCK L_MC4P_GROUPWAITTIME EXTENDS L_MC4P_Template_MoveLicence
VAR_INPUT
	XEXECUTE : BOOL;
	LRTIME : LREAL;
END_VAR
VAR_OUTPUT
	XDONE : BOOL;
	XBUSY : BOOL;
	XACTIVE : BOOL;
	XCOMMANDABORTED : BOOL;
	XERROR : BOOL;
	EERRORID : L_IE1P_Error;
END_VAR
VAR
	WAIT : L_MC4P_GroupWaitTime_Internal;
	PMOVE : POINTER TO L_MC4P_MoveContPath;
END_VAR
END_FUNCTION_BLOCK

(* ---- L_MC4P_GROUPWAITTIME_INTERNAL.pou ---- *)
FUNCTION_BLOCK L_MC4P_GROUPWAITTIME_INTERNAL EXTENDS L_MC4P_MoveContPath
VAR_INPUT
	XEXECUTE : BOOL;
	LRTIME : LREAL;
END_VAR
VAR_OUTPUT
	XDONE : BOOL;
	XBUSY : BOOL;
	XACTIVE : BOOL;
	XCOMMANDABORTED : BOOL;
	XERROR : BOOL;
	EERRORID : L_IE1P_Error;
END_VAR
VAR
	LRTIME_INPUT : LREAL;
	AEAUXMODE : ARRAY [1..6] OF L_MC4P_AuxMode := [6(L_MC4P_AuxMode.Inactive)];
	TRANSITIONPARAMETER : ARRAY [1..12] OF LREAL := [12(0)];
	COORDSYSTEM : L_MC4P_CoordSystem;
	BUFFERMODE : MC_BUFFER_MODE;
	TRANSITIONMODE : MC_TRANSITION_MODE;
	CLASSID : DINT;
END_VAR
END_FUNCTION_BLOCK

METHOD HOMINGREQUIRED : BOOL
END_METHOD

METHOD ISPTP : BOOL
END_METHOD

METHOD MAIN
VAR_IN_OUT
	AXESGROUP : AXES_GROUP_KIN;
	FBBASE : L_MC4P_Template_AG_KIN;
END_VAR
END_METHOD

METHOD PARAMETERFREEZE
VAR_IN_OUT
	AXESGROUP : AXES_GROUP_KIN;
	FBBASE : L_MC4P_Template_AG_KIN;
	COORDSYSTEM : L_MC4P_CoordSystem;
	BUFFERMODE : MC_BUFFER_MODE;
	TRANSITIONMODE : MC_TRANSITION_MODE;
	TRANSITIONPARAMETER : ARRAY [1..12] OF LREAL;
END_VAR
END_METHOD

METHOD SETPATHELEMENT
VAR_IN_OUT
	AXESGROUP : AXES_GROUP_KIN;
	FBBASE : L_MC4P_Template_AG_KIN;
	ALRSTARTPOS : ARRAY [1..12] OF LREAL;
	ALRSUPERPOSPOSATSTART : ARRAY [1..3] OF LREAL;
END_VAR
END_METHOD

(* ---- L_MC4P_INTERPOLATEPATH.pou ---- *)
FUNCTION_BLOCK L_MC4P_INTERPOLATEPATH
VAR_INPUT
	PLIST : POINTER TO L_MC4P_PathDataList;
	PAXESGROUP : POINTER TO AXES_GROUP_KIN;
	XEXCLUDEAUX : BOOL := FALSE;
	XIGNOREOVERRIDEWAITTIME : BOOL := FALSE;
	ITFDIGSWITCHOBSERVER : L_MC4P_IDigSwitchHandling;
END_VAR
VAR_OUTPUT
	AXAUXAXISACTIVE : ARRAY [1..6] OF BOOL;
	NSEGMENTNO : DINT;
	XERROR : BOOL := FALSE;
	EERRORID : L_IE1P_Error;
	DWINTERNALID : DWORD;
END_VAR
VAR
	SCCYCLICDATA : L_MC4P_CyclicData;
	PLISTELEMENTTIME : POINTER TO L_MC4P_ListElement;
	PLISTELEMENTGEO : POINTER TO L_MC4P_ListElement;
	PLISTELEMENTTOBODELETED : POINTER TO L_MC4P_ListElement;
	XREADY : BOOL;
	PATHFILTER : L_MC4P_SetValueFilter;
	AROTFILTER : ARRAY [1..3] OF L_MC4P_SetValueFilter;
	AAUXFILTER : ARRAY [1..6] OF L_MC4P_SetValueFilter;
	EFILTERMODE : L_MC4P_SetValueFilterMode := L_MC4P_SetValueFilterMode.EqualySpaced;
	UIFILTERTIME : UINT;
	XENABLEFILTER : BOOL;
	XAXESGROUPIPOSTANDSTILL : BOOL := TRUE;
	PPAUSEDTIMEELEMENT : POINTER TO L_MC4P_ListElement;
	XPAUSETIMEIPO : BOOL;
	XRELEASETIMEIPO : BOOL;
	AXAUXAXISACTIVEOLD : ARRAY [1..6] OF BOOL;
	XFIRSTCALLOFNEWSEQUENCE : BOOL;
END_VAR
END_FUNCTION_BLOCK

METHOD AXISPASSEDTARGETPOS : BOOL
VAR_INPUT
	ETRAVERSINGRANGE : L_MC1P_TraversingRange;
	LRCYCLELENGTH : LREAL;
	LRSTARTPOS : LREAL;
	LRTARGETPOS : LREAL;
	LRIPOPOS : LREAL;
	LRIPOVEL : LREAL;
	LRIPOACC : LREAL;
	LRIPOPOSOLD : LREAL;
	SCPROFILEDATAACT : REFERENCE TO L_MC1P_ProfileData;
	SCPROFILEDATANEXT : REFERENCE TO L_MC1P_ProfileData;
END_VAR
END_METHOD

METHOD ENDSWITHRESTPHASE : BOOL
VAR_IN_OUT
	PROFILEDATA : L_MC1P_ProfileData;
END_VAR
END_METHOD

METHOD GEOMETRYPASSED : BOOL
VAR_IN_OUT
	PLISTELEMENT : POINTER TO L_MC4P_ListElement;
	SCCYCLICDATA : L_MC4P_CyclicData;
END_VAR
END_METHOD

METHOD GETSTARTDIRECTION : MC_Direction
VAR_IN_OUT
	PROFILEDATA : L_MC1P_ProfileData;
END_VAR
END_METHOD

METHOD GETTARGETDIRECTION : MC_Direction
VAR_IN_OUT
	PROFILEDATA : L_MC1P_ProfileData;
END_VAR
END_METHOD

METHOD INITIPO
END_METHOD

METHOD INTERPOLATECPGEOMETRY
VAR_IN_OUT
	PLISTELEMENTGEO : POINTER TO L_MC4P_ListElement;
	SCCYCLICDATA : L_MC4P_CyclicData;
END_VAR
END_METHOD

METHOD INTERPOLATETIMEPROFILES
VAR_IN_OUT
	PLISTELEMENTTIME : POINTER TO L_MC4P_ListElement;
	SCCYCLICDATA : L_MC4P_CyclicData;
END_VAR
END_METHOD

METHOD INTERPOLATOR
VAR_IN_OUT
	PLISTELEMENTTIME : POINTER TO L_MC4P_ListElement;
	PLISTELEMENTGEO : POINTER TO L_MC4P_ListElement;
	SCCYCLICDATA : L_MC4P_CyclicData;
END_VAR
END_METHOD

METHOD ISCARTESIAN : BOOL
VAR_INPUT
	ESEGMENTTYPE : L_MC4P_SegmentType;
END_VAR
END_METHOD

METHOD MODULOFILTEROVERRIDE
VAR_IN_OUT
	PLISTELEMENTTIME : POINTER TO L_MC4P_ListElement;
	SCCYCLICDATA : L_MC4P_CyclicData;
END_VAR
END_METHOD

METHOD RESETIPO
END_METHOD

METHOD TARGETVELOFLISTELEMENTEQ0 : BOOL
VAR_INPUT
	PLISTELEMENT : POINTER TO L_MC4P_ListElement;
END_VAR
END_METHOD
